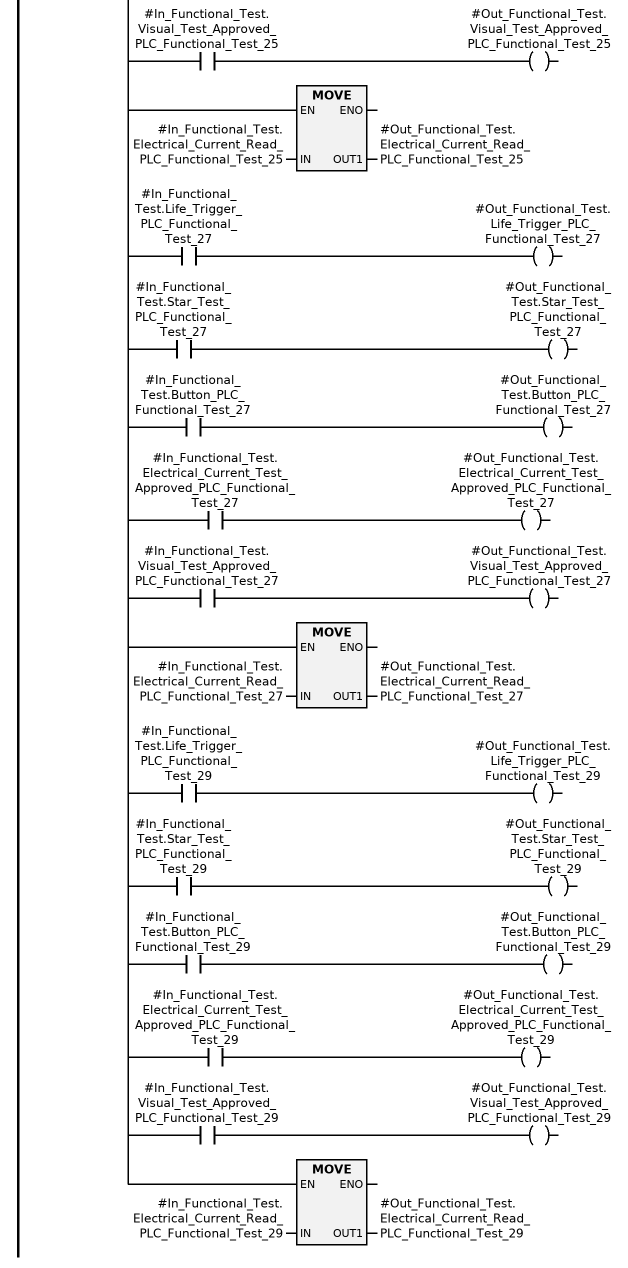
   RUNG wire#powerrail
      { S7_Templates := "SrcType := SInt" } EQ_Contact(in1 := #Test_Station, in2 := 7)
      wire#w1
      Contact( #Life_Trigger )
      Coil( #Out_Functional_Test.Life_Trigger_PLC_Functional_Test_7 )
   END_RUNG
   RUNG wire#w1
      Contact( #Star_Test )
      Coil( #Out_Functional_Test.Star_Test_PLC_Functional_Test_7 )
   END_RUNG
   RUNG wire#w1
      Contact( #Button_Start_Approve )
      Coil( #Out_Functional_Test.Button_PLC_Functional_Test_7 )
   END_RUNG
   RUNG wire#w1
      Contact( #Electrical_Current_Test_Approved )
      Coil( #Out_Functional_Test.Electrical_Current_Test_Approved_PLC_Functional_Test_7 )
   END_RUNG
   RUNG wire#w1
      Contact( #Visual_Test_Approved )
      Coil( #Out_Functional_Test.Visual_Test_Approved_PLC_Functional_Test_7 )
   END_RUNG
   RUNG wire#w1
      Contact( #In_Test_Parameters.Reset_PLC_Functional_Test_7 )
      Coil( #Reset_Functional_Test )
   END_RUNG
   RUNG wire#w1
      Move(in := #Electrical_Current_Read, out1 => #Out_Functional_Test.Electrical_Current_Read_PLC_Functional_Test_7)
   END_RUNG
   RUNG wire#w1
      Contact( #In_Functional_Test.Life_Trigger_PLC_Functional_Test_9 )
      Coil( #Out_Functional_Test.Life_Trigger_PLC_Functional_Test_9 )
   END_RUNG
   RUNG wire#w1
      Contact( #In_Functional_Test.Star_Test_PLC_Functional_Test_9 )
      Coil( #Out_Functional_Test.Star_Test_PLC_Functional_Test_9 )
   END_RUNG
   RUNG wire#w1
      Contact( #In_Functional_Test.Button_PLC_Functional_Test_9 )
      Coil( #Out_Functional_Test.Button_PLC_Functional_Test_9 )
   END_RUNG
   RUNG wire#w1
      Contact( #In_Functional_Test.Electrical_Current_Test_Approved_PLC_Functional_Test_9 )
      Coil( #Out_Functional_Test.Electrical_Current_Test_Approved_PLC_Functional_Test_9 )
   END_RUNG
   RUNG wire#w1
      Contact( #In_Functional_Test.Visual_Test_Approved_PLC_Functional_Test_9 )
      Coil( #Out_Functional_Test.Visual_Test_Approved_PLC_Functional_Test_9 )
   END_RUNG
   RUNG wire#w1
      Move(in := #In_Functional_Test.Electrical_Current_Read_PLC_Functional_Test_9, out1 => #Out_Functional_Test.Electrical_Current_Read_PLC_Functional_Test_9)
   END_RUNG
   RUNG wire#w1
      Contact( #In_Functional_Test.Life_Trigger_PLC_Functional_Test_11 )
      Coil( #Out_Functional_Test.Life_Trigger_PLC_Functional_Test_11 )
   END_RUNG
   RUNG wire#w1
      Contact( #In_Functional_Test.Star_Test_PLC_Functional_Test_11 )
      Coil( #Out_Functional_Test.Star_Test_PLC_Functional_Test_11 )
   END_RUNG
   RUNG wire#w1
      Contact( #In_Functional_Test.Button_PLC_Functional_Test_11 )
      Coil( #Out_Functional_Test.Button_PLC_Functional_Test_11 )
   END_RUNG
   RUNG wire#w1
      Contact( #In_Functional_Test.Electrical_Current_Test_Approved_PLC_Functional_Test_11 )
      Coil( #Out_Functional_Test.Electrical_Current_Test_Approved_PLC_Functional_Test_11 )
   END_RUNG
   RUNG wire#w1
      Contact( #In_Functional_Test.Visual_Test_Approved_PLC_Functional_Test_11 )
      Coil( #Out_Functional_Test.Visual_Test_Approved_PLC_Functional_Test_11 )
   END_RUNG
   RUNG wire#w1
      Move(in := #In_Functional_Test.Electrical_Current_Read_PLC_Functional_Test_11, out1 => #Out_Functional_Test.Electrical_Current_Read_PLC_Functional_Test_11)
   END_RUNG
   RUNG wire#w1
      Contact( #In_Functional_Test.Life_Trigger_PLC_Functional_Test_13 )
      Coil( #Out_Functional_Test.Life_Trigger_PLC_Functional_Test_13 )
   END_RUNG
   RUNG wire#w1
      Contact( #In_Functional_Test.Star_Test_PLC_Functional_Test_13 )
      Coil( #Out_Functional_Test.Star_Test_PLC_Functional_Test_13 )
   END_RUNG
   RUNG wire#w1
      Contact( #In_Functional_Test.Button_PLC_Functional_Test_13 )
      Coil( #Out_Functional_Test.Button_PLC_Functional_Test_13 )
   END_RUNG
   RUNG wire#w1
      Contact( #In_Functional_Test.Electrical_Current_Test_Approved_PLC_Functional_Test_13 )
      Coil( #Out_Functional_Test.Electrical_Current_Test_Approved_PLC_Functional_Test_13 )
   END_RUNG
   RUNG wire#w1
      Contact( #In_Functional_Test.Visual_Test_Approved_PLC_Functional_Test_13 )
      Coil( #Out_Functional_Test.Visual_Test_Approved_PLC_Functional_Test_13 )
   END_RUNG
   RUNG wire#w1
      Move(in := #In_Functional_Test.Electrical_Current_Read_PLC_Functional_Test_13, out1 => #Out_Functional_Test.Electrical_Current_Read_PLC_Functional_Test_13)
   END_RUNG
   RUNG wire#w1
      Contact( #In_Functional_Test.Life_Trigger_PLC_Functional_Test_15 )
      Coil( #Out_Functional_Test.Life_Trigger_PLC_Functional_Test_15 )
   END_RUNG
   RUNG wire#w1
      Contact( #In_Functional_Test.Star_Test_PLC_Functional_Test_15 )
      Coil( #Out_Functional_Test.Star_Test_PLC_Functional_Test_15 )
   END_RUNG
   RUNG wire#w1
      Contact( #In_Functional_Test.Button_PLC_Functional_Test_15 )
      Coil( #Out_Functional_Test.Button_PLC_Functional_Test_15 )
   END_RUNG
   RUNG wire#w1
      Contact( #In_Functional_Test.Electrical_Current_Test_Approved_PLC_Functional_Test_15 )
      Coil( #Out_Functional_Test.Electrical_Current_Test_Approved_PLC_Functional_Test_15 )
   END_RUNG
   RUNG wire#w1
      Contact( #In_Functional_Test.Visual_Test_Approved_PLC_Functional_Test_15 )
      Coil( #Out_Functional_Test.Visual_Test_Approved_PLC_Functional_Test_15 )
   END_RUNG
   RUNG wire#w1
      Move(in := #In_Functional_Test.Electrical_Current_Read_PLC_Functional_Test_15, out1 => #Out_Functional_Test.Electrical_Current_Read_PLC_Functional_Test_15)
   END_RUNG
   RUNG wire#w1
      Contact( #In_Functional_Test.Life_Trigger_PLC_Functional_Test_17 )
      Coil( #Out_Functional_Test.Life_Trigger_PLC_Functional_Test_17 )
   END_RUNG
   RUNG wire#w1
      Contact( #In_Functional_Test.Star_Test_PLC_Functional_Test_17 )
      Coil( #Out_Functional_Test.Star_Test_PLC_Functional_Test_17 )
   END_RUNG
   RUNG wire#w1
      Contact( #In_Functional_Test.Button_PLC_Functional_Test_17 )
      Coil( #Out_Functional_Test.Button_PLC_Functional_Test_17 )
   END_RUNG
   RUNG wire#w1
      Contact( #In_Functional_Test.Electrical_Current_Test_Approved_PLC_Functional_Test_17 )
      Coil( #Out_Functional_Test.Electrical_Current_Test_Approved_PLC_Functional_Test_17 )
   END_RUNG
   RUNG wire#w1
      Contact( #In_Functional_Test.Visual_Test_Approved_PLC_Functional_Test_17 )
      Coil( #Out_Functional_Test.Visual_Test_Approved_PLC_Functional_Test_17 )
   END_RUNG
   RUNG wire#w1
      Move(in := #In_Functional_Test.Electrical_Current_Read_PLC_Functional_Test_17, out1 => #Out_Functional_Test.Electrical_Current_Read_PLC_Functional_Test_17)
   END_RUNG
   RUNG wire#w1
      Contact( #In_Functional_Test.Life_Trigger_PLC_Functional_Test_19 )
      Coil( #Out_Functional_Test.Life_Trigger_PLC_Functional_Test_19 )
   END_RUNG
   RUNG wire#w1
      Contact( #In_Functional_Test.Star_Test_PLC_Functional_Test_19 )
      Coil( #Out_Functional_Test.Star_Test_PLC_Functional_Test_19 )
   END_RUNG
   RUNG wire#w1
      Contact( #In_Functional_Test.Button_PLC_Functional_Test_19 )
      Coil( #Out_Functional_Test.Button_PLC_Functional_Test_19 )
   END_RUNG
   RUNG wire#w1
      Contact( #In_Functional_Test.Electrical_Current_Test_Approved_PLC_Functional_Test_19 )
      Coil( #Out_Functional_Test.Electrical_Current_Test_Approved_PLC_Functional_Test_19 )
   END_RUNG
   RUNG wire#w1
      Contact( #In_Functional_Test.Visual_Test_Approved_PLC_Functional_Test_19 )
      Coil( #Out_Functional_Test.Visual_Test_Approved_PLC_Functional_Test_19 )
   END_RUNG
   RUNG wire#w1
      Move(in := #In_Functional_Test.Electrical_Current_Read_PLC_Functional_Test_19, out1 => #Out_Functional_Test.Electrical_Current_Read_PLC_Functional_Test_19)
   END_RUNG
   RUNG wire#w1
      Contact( #In_Functional_Test.Life_Trigger_PLC_Functional_Test_21 )
      Coil( #Out_Functional_Test.Life_Trigger_PLC_Functional_Test_21 )
   END_RUNG
   RUNG wire#w1
      Contact( #In_Functional_Test.Star_Test_PLC_Functional_Test_21 )
      Coil( #Out_Functional_Test.Star_Test_PLC_Functional_Test_21 )
   END_RUNG
   RUNG wire#w1
      Contact( #In_Functional_Test.Button_PLC_Functional_Test_21 )
      Coil( #Out_Functional_Test.Button_PLC_Functional_Test_21 )
   END_RUNG
   RUNG wire#w1
      Contact( #In_Functional_Test.Electrical_Current_Test_Approved_PLC_Functional_Test_21 )
      Coil( #Out_Functional_Test.Electrical_Current_Test_Approved_PLC_Functional_Test_21 )
   END_RUNG
   RUNG wire#w1
      Contact( #In_Functional_Test.Visual_Test_Approved_PLC_Functional_Test_21 )
      Coil( #Out_Functional_Test.Visual_Test_Approved_PLC_Functional_Test_21 )
   END_RUNG
   RUNG wire#w1
      Move(in := #In_Functional_Test.Electrical_Current_Read_PLC_Functional_Test_21, out1 => #Out_Functional_Test.Electrical_Current_Read_PLC_Functional_Test_21)
   END_RUNG
   RUNG wire#w1
      Contact( #In_Functional_Test.Life_Trigger_PLC_Functional_Test_23 )
      Coil( #Out_Functional_Test.Life_Trigger_PLC_Functional_Test_23 )
   END_RUNG
   RUNG wire#w1
      Contact( #In_Functional_Test.Star_Test_PLC_Functional_Test_23 )
      Coil( #Out_Functional_Test.Star_Test_PLC_Functional_Test_23 )
   END_RUNG
   RUNG wire#w1
      Contact( #In_Functional_Test.Button_PLC_Functional_Test_23 )
      Coil( #Out_Functional_Test.Button_PLC_Functional_Test_23 )
   END_RUNG
   RUNG wire#w1
      Contact( #In_Functional_Test.Electrical_Current_Test_Approved_PLC_Functional_Test_23 )
      Coil( #Out_Functional_Test.Electrical_Current_Test_Approved_PLC_Functional_Test_23 )
   END_RUNG
   RUNG wire#w1
      Contact( #In_Functional_Test.Visual_Test_Approved_PLC_Functional_Test_23 )
      Coil( #Out_Functional_Test.Visual_Test_Approved_PLC_Functional_Test_23 )
   END_RUNG
   RUNG wire#w1
      Move(in := #In_Functional_Test.Electrical_Current_Read_PLC_Functional_Test_23, out1 => #Out_Functional_Test.Electrical_Current_Read_PLC_Functional_Test_23)
   END_RUNG
   RUNG wire#w1
      Contact( #In_Functional_Test.Life_Trigger_PLC_Functional_Test_25 )
      Coil( #Out_Functional_Test.Life_Trigger_PLC_Functional_Test_25 )
   END_RUNG
   RUNG wire#w1
      Contact( #In_Functional_Test.Star_Test_PLC_Functional_Test_25 )
      Coil( #Out_Functional_Test.Star_Test_PLC_Functional_Test_25 )
   END_RUNG
   RUNG wire#w1
      Contact( #In_Functional_Test.Button_PLC_Functional_Test_25 )
      Coil( #Out_Functional_Test.Button_PLC_Functional_Test_25 )
   END_RUNG
   RUNG wire#w1
      Contact( #In_Functional_Test.Electrical_Current_Test_Approved_PLC_Functional_Test_25 )
      Coil( #Out_Functional_Test.Electrical_Current_Test_Approved_PLC_Functional_Test_25 )
   END_RUNG
   RUNG wire#w1
      Contact( #In_Functional_Test.Visual_Test_Approved_PLC_Functional_Test_25 )
      Coil( #Out_Functional_Test.Visual_Test_Approved_PLC_Functional_Test_25 )
   END_RUNG
   RUNG wire#w1
      Move(in := #In_Functional_Test.Electrical_Current_Read_PLC_Functional_Test_25, out1 => #Out_Functional_Test.Electrical_Current_Read_PLC_Functional_Test_25)
   END_RUNG
   RUNG wire#w1
      Contact( #In_Functional_Test.Life_Trigger_PLC_Functional_Test_27 )
      Coil( #Out_Functional_Test.Life_Trigger_PLC_Functional_Test_27 )
   END_RUNG
   RUNG wire#w1
      Contact( #In_Functional_Test.Star_Test_PLC_Functional_Test_27 )
      Coil( #Out_Functional_Test.Star_Test_PLC_Functional_Test_27 )
   END_RUNG
   RUNG wire#w1
      Contact( #In_Functional_Test.Button_PLC_Functional_Test_27 )
      Coil( #Out_Functional_Test.Button_PLC_Functional_Test_27 )
   END_RUNG
   RUNG wire#w1
      Contact( #In_Functional_Test.Electrical_Current_Test_Approved_PLC_Functional_Test_27 )
      Coil( #Out_Functional_Test.Electrical_Current_Test_Approved_PLC_Functional_Test_27 )
   END_RUNG
   RUNG wire#w1
      Contact( #In_Functional_Test.Visual_Test_Approved_PLC_Functional_Test_27 )
      Coil( #Out_Functional_Test.Visual_Test_Approved_PLC_Functional_Test_27 )
   END_RUNG
   RUNG wire#w1
      Move(in := #In_Functional_Test.Electrical_Current_Read_PLC_Functional_Test_27, out1 => #Out_Functional_Test.Electrical_Current_Read_PLC_Functional_Test_27)
   END_RUNG
   RUNG wire#w1
      Contact( #In_Functional_Test.Life_Trigger_PLC_Functional_Test_29 )
      Coil( #Out_Functional_Test.Life_Trigger_PLC_Functional_Test_29 )
   END_RUNG
   RUNG wire#w1
      Contact( #In_Functional_Test.Star_Test_PLC_Functional_Test_29 )
      Coil( #Out_Functional_Test.Star_Test_PLC_Functional_Test_29 )
   END_RUNG
   RUNG wire#w1
      Contact( #In_Functional_Test.Button_PLC_Functional_Test_29 )
      Coil( #Out_Functional_Test.Button_PLC_Functional_Test_29 )
   END_RUNG
   RUNG wire#w1
      Contact( #In_Functional_Test.Electrical_Current_Test_Approved_PLC_Functional_Test_29 )
      Coil( #Out_Functional_Test.Electrical_Current_Test_Approved_PLC_Functional_Test_29 )
   END_RUNG
   RUNG wire#w1
      Contact( #In_Functional_Test.Visual_Test_Approved_PLC_Functional_Test_29 )
      Coil( #Out_Functional_Test.Visual_Test_Approved_PLC_Functional_Test_29 )
   END_RUNG
   RUNG wire#w1
      Move(in := #In_Functional_Test.Electrical_Current_Read_PLC_Functional_Test_29, out1 => #Out_Functional_Test.Electrical_Current_Read_PLC_Functional_Test_29)
   END_RUNG
   // the same network as SCL:
   #_w1 := #Test_Station = 7;
   #Out_Functional_Test.Life_Trigger_PLC_Functional_Test_7 := #_w1 AND #Life_Trigger;
   #Out_Functional_Test.Star_Test_PLC_Functional_Test_7 := #_w1 AND #Star_Test;
   #Out_Functional_Test.Button_PLC_Functional_Test_7 := #_w1 AND #Button_Start_Approve;
   #Out_Functional_Test.Electrical_Current_Test_Approved_PLC_Functional_Test_7 := #_w1 AND #Electrical_Current_Test_Approved;
   #Out_Functional_Test.Visual_Test_Approved_PLC_Functional_Test_7 := #_w1 AND #Visual_Test_Approved;
   #Reset_Functional_Test := #_w1 AND #In_Test_Parameters.Reset_PLC_Functional_Test_7;
   IF #_w1 THEN
       #Out_Functional_Test.Electrical_Current_Read_PLC_Functional_Test_7 := #Electrical_Current_Read;
   END_IF;
   #Out_Functional_Test.Life_Trigger_PLC_Functional_Test_9 := #_w1 AND #In_Functional_Test.Life_Trigger_PLC_Functional_Test_9;
   #Out_Functional_Test.Star_Test_PLC_Functional_Test_9 := #_w1 AND #In_Functional_Test.Star_Test_PLC_Functional_Test_9;
   #Out_Functional_Test.Button_PLC_Functional_Test_9 := #_w1 AND #In_Functional_Test.Button_PLC_Functional_Test_9;
   #Out_Functional_Test.Electrical_Current_Test_Approved_PLC_Functional_Test_9 := #_w1 AND #In_Functional_Test.Electrical_Current_Test_Approved_PLC_Functional_Test_9;
   #Out_Functional_Test.Visual_Test_Approved_PLC_Functional_Test_9 := #_w1 AND #In_Functional_Test.Visual_Test_Approved_PLC_Functional_Test_9;
   IF #_w1 THEN
       #Out_Functional_Test.Electrical_Current_Read_PLC_Functional_Test_9 := #In_Functional_Test.Electrical_Current_Read_PLC_Functional_Test_9;
   END_IF;
   #Out_Functional_Test.Life_Trigger_PLC_Functional_Test_11 := #_w1 AND #In_Functional_Test.Life_Trigger_PLC_Functional_Test_11;
   #Out_Functional_Test.Star_Test_PLC_Functional_Test_11 := #_w1 AND #In_Functional_Test.Star_Test_PLC_Functional_Test_11;
   #Out_Functional_Test.Button_PLC_Functional_Test_11 := #_w1 AND #In_Functional_Test.Button_PLC_Functional_Test_11;
   #Out_Functional_Test.Electrical_Current_Test_Approved_PLC_Functional_Test_11 := #_w1 AND #In_Functional_Test.Electrical_Current_Test_Approved_PLC_Functional_Test_11;
   #Out_Functional_Test.Visual_Test_Approved_PLC_Functional_Test_11 := #_w1 AND #In_Functional_Test.Visual_Test_Approved_PLC_Functional_Test_11;
   IF #_w1 THEN
       #Out_Functional_Test.Electrical_Current_Read_PLC_Functional_Test_11 := #In_Functional_Test.Electrical_Current_Read_PLC_Functional_Test_11;
   END_IF;
   #Out_Functional_Test.Life_Trigger_PLC_Functional_Test_13 := #_w1 AND #In_Functional_Test.Life_Trigger_PLC_Functional_Test_13;
   #Out_Functional_Test.Star_Test_PLC_Functional_Test_13 := #_w1 AND #In_Functional_Test.Star_Test_PLC_Functional_Test_13;
   #Out_Functional_Test.Button_PLC_Functional_Test_13 := #_w1 AND #In_Functional_Test.Button_PLC_Functional_Test_13;
   #Out_Functional_Test.Electrical_Current_Test_Approved_PLC_Functional_Test_13 := #_w1 AND #In_Functional_Test.Electrical_Current_Test_Approved_PLC_Functional_Test_13;
   #Out_Functional_Test.Visual_Test_Approved_PLC_Functional_Test_13 := #_w1 AND #In_Functional_Test.Visual_Test_Approved_PLC_Functional_Test_13;
   IF #_w1 THEN
       #Out_Functional_Test.Electrical_Current_Read_PLC_Functional_Test_13 := #In_Functional_Test.Electrical_Current_Read_PLC_Functional_Test_13;
   END_IF;
   #Out_Functional_Test.Life_Trigger_PLC_Functional_Test_15 := #_w1 AND #In_Functional_Test.Life_Trigger_PLC_Functional_Test_15;
   #Out_Functional_Test.Star_Test_PLC_Functional_Test_15 := #_w1 AND #In_Functional_Test.Star_Test_PLC_Functional_Test_15;
   #Out_Functional_Test.Button_PLC_Functional_Test_15 := #_w1 AND #In_Functional_Test.Button_PLC_Functional_Test_15;
   #Out_Functional_Test.Electrical_Current_Test_Approved_PLC_Functional_Test_15 := #_w1 AND #In_Functional_Test.Electrical_Current_Test_Approved_PLC_Functional_Test_15;
   #Out_Functional_Test.Visual_Test_Approved_PLC_Functional_Test_15 := #_w1 AND #In_Functional_Test.Visual_Test_Approved_PLC_Functional_Test_15;
   IF #_w1 THEN
       #Out_Functional_Test.Electrical_Current_Read_PLC_Functional_Test_15 := #In_Functional_Test.Electrical_Current_Read_PLC_Functional_Test_15;
   END_IF;
   #Out_Functional_Test.Life_Trigger_PLC_Functional_Test_17 := #_w1 AND #In_Functional_Test.Life_Trigger_PLC_Functional_Test_17;
   #Out_Functional_Test.Star_Test_PLC_Functional_Test_17 := #_w1 AND #In_Functional_Test.Star_Test_PLC_Functional_Test_17;
   #Out_Functional_Test.Button_PLC_Functional_Test_17 := #_w1 AND #In_Functional_Test.Button_PLC_Functional_Test_17;
   #Out_Functional_Test.Electrical_Current_Test_Approved_PLC_Functional_Test_17 := #_w1 AND #In_Functional_Test.Electrical_Current_Test_Approved_PLC_Functional_Test_17;
   #Out_Functional_Test.Visual_Test_Approved_PLC_Functional_Test_17 := #_w1 AND #In_Functional_Test.Visual_Test_Approved_PLC_Functional_Test_17;
   IF #_w1 THEN
       #Out_Functional_Test.Electrical_Current_Read_PLC_Functional_Test_17 := #In_Functional_Test.Electrical_Current_Read_PLC_Functional_Test_17;
   END_IF;
   #Out_Functional_Test.Life_Trigger_PLC_Functional_Test_19 := #_w1 AND #In_Functional_Test.Life_Trigger_PLC_Functional_Test_19;
   #Out_Functional_Test.Star_Test_PLC_Functional_Test_19 := #_w1 AND #In_Functional_Test.Star_Test_PLC_Functional_Test_19;
   #Out_Functional_Test.Button_PLC_Functional_Test_19 := #_w1 AND #In_Functional_Test.Button_PLC_Functional_Test_19;
   #Out_Functional_Test.Electrical_Current_Test_Approved_PLC_Functional_Test_19 := #_w1 AND #In_Functional_Test.Electrical_Current_Test_Approved_PLC_Functional_Test_19;
   #Out_Functional_Test.Visual_Test_Approved_PLC_Functional_Test_19 := #_w1 AND #In_Functional_Test.Visual_Test_Approved_PLC_Functional_Test_19;
   IF #_w1 THEN
       #Out_Functional_Test.Electrical_Current_Read_PLC_Functional_Test_19 := #In_Functional_Test.Electrical_Current_Read_PLC_Functional_Test_19;
   END_IF;
   #Out_Functional_Test.Life_Trigger_PLC_Functional_Test_21 := #_w1 AND #In_Functional_Test.Life_Trigger_PLC_Functional_Test_21;
   #Out_Functional_Test.Star_Test_PLC_Functional_Test_21 := #_w1 AND #In_Functional_Test.Star_Test_PLC_Functional_Test_21;
   #Out_Functional_Test.Button_PLC_Functional_Test_21 := #_w1 AND #In_Functional_Test.Button_PLC_Functional_Test_21;
   #Out_Functional_Test.Electrical_Current_Test_Approved_PLC_Functional_Test_21 := #_w1 AND #In_Functional_Test.Electrical_Current_Test_Approved_PLC_Functional_Test_21;
   #Out_Functional_Test.Visual_Test_Approved_PLC_Functional_Test_21 := #_w1 AND #In_Functional_Test.Visual_Test_Approved_PLC_Functional_Test_21;
   IF #_w1 THEN
       #Out_Functional_Test.Electrical_Current_Read_PLC_Functional_Test_21 := #In_Functional_Test.Electrical_Current_Read_PLC_Functional_Test_21;
   END_IF;
   #Out_Functional_Test.Life_Trigger_PLC_Functional_Test_23 := #_w1 AND #In_Functional_Test.Life_Trigger_PLC_Functional_Test_23;
   #Out_Functional_Test.Star_Test_PLC_Functional_Test_23 := #_w1 AND #In_Functional_Test.Star_Test_PLC_Functional_Test_23;
   #Out_Functional_Test.Button_PLC_Functional_Test_23 := #_w1 AND #In_Functional_Test.Button_PLC_Functional_Test_23;
   #Out_Functional_Test.Electrical_Current_Test_Approved_PLC_Functional_Test_23 := #_w1 AND #In_Functional_Test.Electrical_Current_Test_Approved_PLC_Functional_Test_23;
   #Out_Functional_Test.Visual_Test_Approved_PLC_Functional_Test_23 := #_w1 AND #In_Functional_Test.Visual_Test_Approved_PLC_Functional_Test_23;
   IF #_w1 THEN
       #Out_Functional_Test.Electrical_Current_Read_PLC_Functional_Test_23 := #In_Functional_Test.Electrical_Current_Read_PLC_Functional_Test_23;
   END_IF;
   #Out_Functional_Test.Life_Trigger_PLC_Functional_Test_25 := #_w1 AND #In_Functional_Test.Life_Trigger_PLC_Functional_Test_25;
   #Out_Functional_Test.Star_Test_PLC_Functional_Test_25 := #_w1 AND #In_Functional_Test.Star_Test_PLC_Functional_Test_25;
   #Out_Functional_Test.Button_PLC_Functional_Test_25 := #_w1 AND #In_Functional_Test.Button_PLC_Functional_Test_25;
   #Out_Functional_Test.Electrical_Current_Test_Approved_PLC_Functional_Test_25 := #_w1 AND #In_Functional_Test.Electrical_Current_Test_Approved_PLC_Functional_Test_25;
   #Out_Functional_Test.Visual_Test_Approved_PLC_Functional_Test_25 := #_w1 AND #In_Functional_Test.Visual_Test_Approved_PLC_Functional_Test_25;
   IF #_w1 THEN
       #Out_Functional_Test.Electrical_Current_Read_PLC_Functional_Test_25 := #In_Functional_Test.Electrical_Current_Read_PLC_Functional_Test_25;
   END_IF;
   #Out_Functional_Test.Life_Trigger_PLC_Functional_Test_27 := #_w1 AND #In_Functional_Test.Life_Trigger_PLC_Functional_Test_27;
   #Out_Functional_Test.Star_Test_PLC_Functional_Test_27 := #_w1 AND #In_Functional_Test.Star_Test_PLC_Functional_Test_27;
   #Out_Functional_Test.Button_PLC_Functional_Test_27 := #_w1 AND #In_Functional_Test.Button_PLC_Functional_Test_27;
   #Out_Functional_Test.Electrical_Current_Test_Approved_PLC_Functional_Test_27 := #_w1 AND #In_Functional_Test.Electrical_Current_Test_Approved_PLC_Functional_Test_27;
   #Out_Functional_Test.Visual_Test_Approved_PLC_Functional_Test_27 := #_w1 AND #In_Functional_Test.Visual_Test_Approved_PLC_Functional_Test_27;
   IF #_w1 THEN
       #Out_Functional_Test.Electrical_Current_Read_PLC_Functional_Test_27 := #In_Functional_Test.Electrical_Current_Read_PLC_Functional_Test_27;
   END_IF;
   #Out_Functional_Test.Life_Trigger_PLC_Functional_Test_29 := #_w1 AND #In_Functional_Test.Life_Trigger_PLC_Functional_Test_29;
   #Out_Functional_Test.Star_Test_PLC_Functional_Test_29 := #_w1 AND #In_Functional_Test.Star_Test_PLC_Functional_Test_29;
   #Out_Functional_Test.Button_PLC_Functional_Test_29 := #_w1 AND #In_Functional_Test.Button_PLC_Functional_Test_29;
   #Out_Functional_Test.Electrical_Current_Test_Approved_PLC_Functional_Test_29 := #_w1 AND #In_Functional_Test.Electrical_Current_Test_Approved_PLC_Functional_Test_29;
   #Out_Functional_Test.Visual_Test_Approved_PLC_Functional_Test_29 := #_w1 AND #In_Functional_Test.Visual_Test_Approved_PLC_Functional_Test_29;
   IF #_w1 THEN
       #Out_Functional_Test.Electrical_Current_Read_PLC_Functional_Test_29 := #In_Functional_Test.Electrical_Current_Read_PLC_Functional_Test_29;
   END_IF;
END_REGION

REGION Network 6: Functional Test Station 9
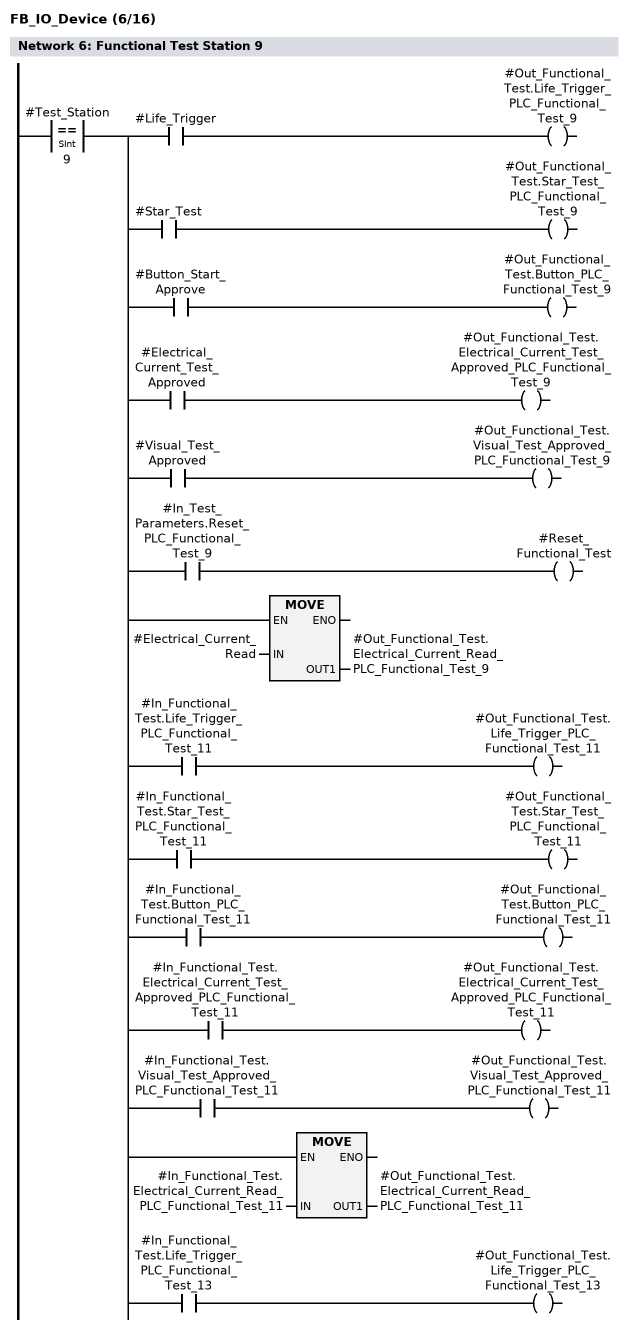
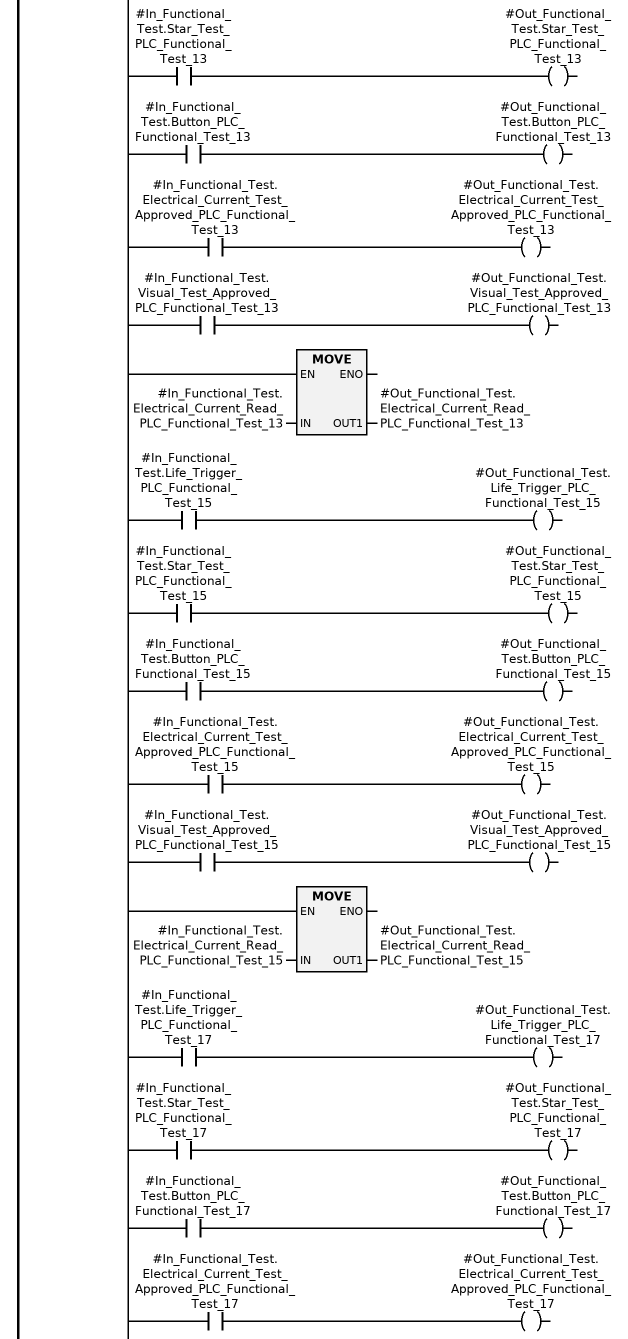
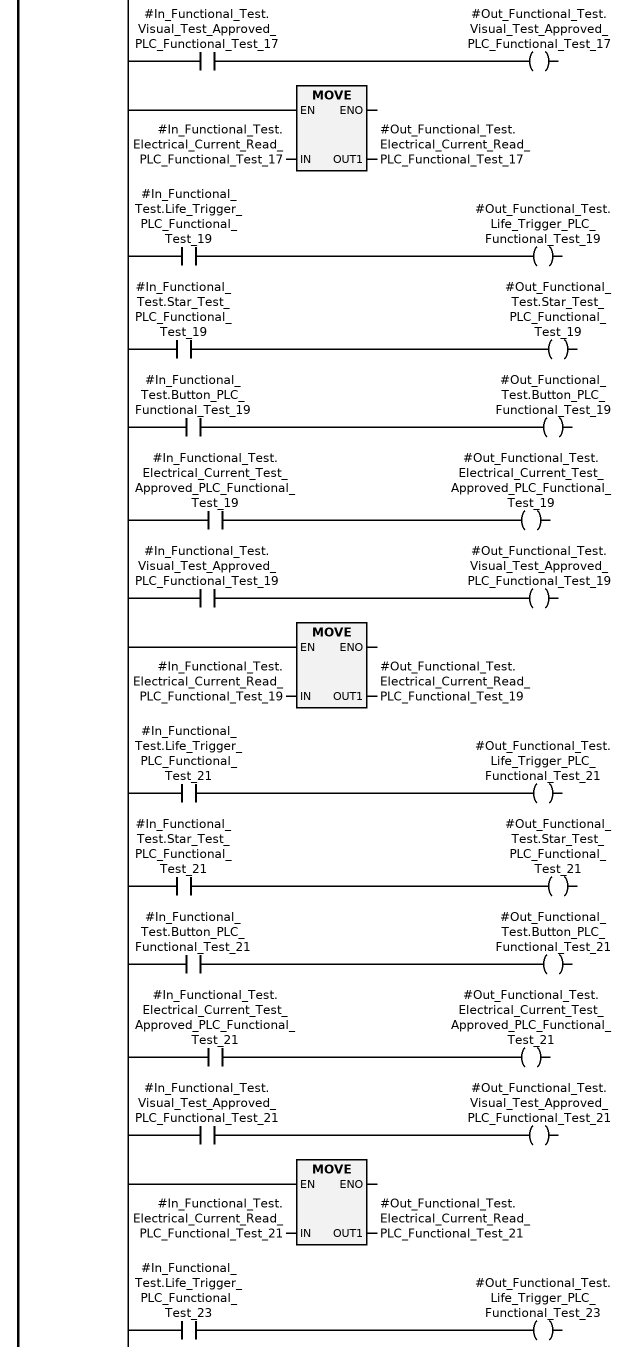
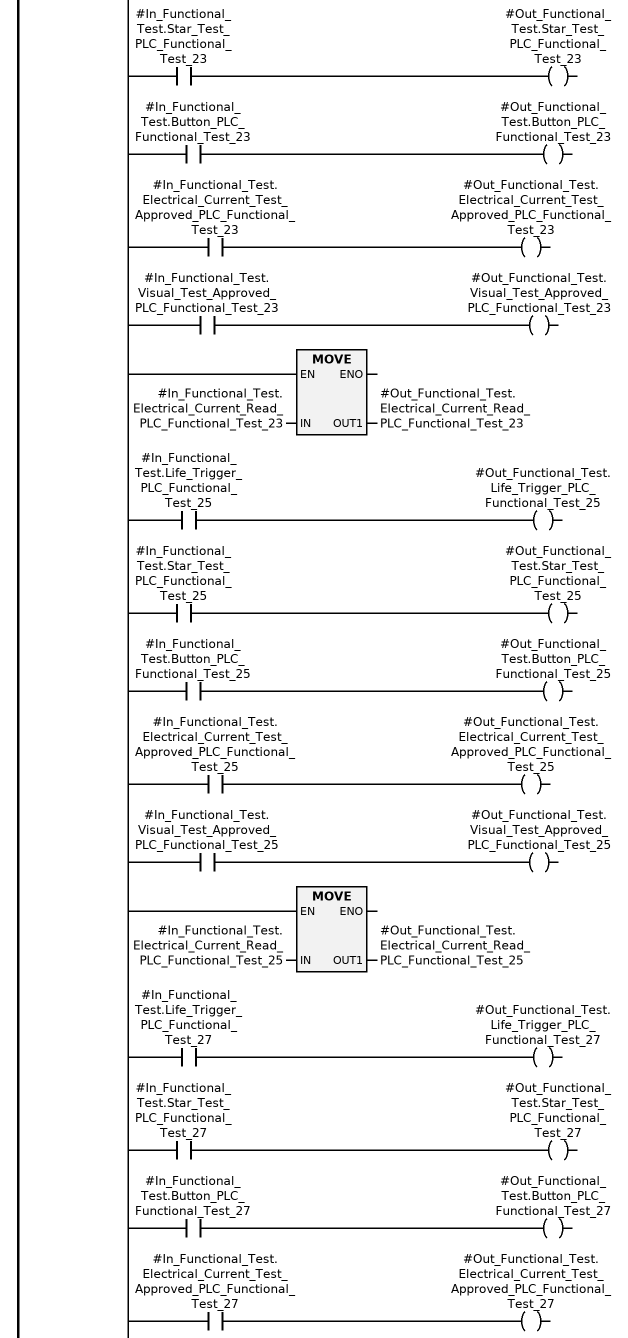
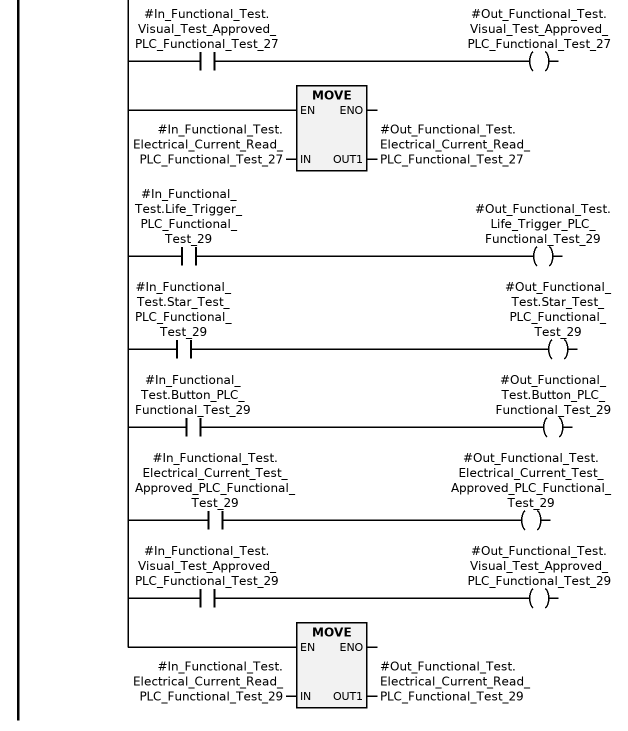
   RUNG wire#powerrail
      { S7_Templates := "SrcType := SInt" } EQ_Contact(in1 := #Test_Station, in2 := 9)
      wire#w1
      Contact( #Life_Trigger )
      Coil( #Out_Functional_Test.Life_Trigger_PLC_Functional_Test_9 )
   END_RUNG
   RUNG wire#w1
      Contact( #Star_Test )
      Coil( #Out_Functional_Test.Star_Test_PLC_Functional_Test_9 )
   END_RUNG
   RUNG wire#w1
      Contact( #Button_Start_Approve )
      Coil( #Out_Functional_Test.Button_PLC_Functional_Test_9 )
   END_RUNG
   RUNG wire#w1
      Contact( #Electrical_Current_Test_Approved )
      Coil( #Out_Functional_Test.Electrical_Current_Test_Approved_PLC_Functional_Test_9 )
   END_RUNG
   RUNG wire#w1
      Contact( #Visual_Test_Approved )
      Coil( #Out_Functional_Test.Visual_Test_Approved_PLC_Functional_Test_9 )
   END_RUNG
   RUNG wire#w1
      Contact( #In_Test_Parameters.Reset_PLC_Functional_Test_9 )
      Coil( #Reset_Functional_Test )
   END_RUNG
   RUNG wire#w1
      Move(in := #Electrical_Current_Read, out1 => #Out_Functional_Test.Electrical_Current_Read_PLC_Functional_Test_9)
   END_RUNG
   RUNG wire#w1
      Contact( #In_Functional_Test.Life_Trigger_PLC_Functional_Test_11 )
      Coil( #Out_Functional_Test.Life_Trigger_PLC_Functional_Test_11 )
   END_RUNG
   RUNG wire#w1
      Contact( #In_Functional_Test.Star_Test_PLC_Functional_Test_11 )
      Coil( #Out_Functional_Test.Star_Test_PLC_Functional_Test_11 )
   END_RUNG
   RUNG wire#w1
      Contact( #In_Functional_Test.Button_PLC_Functional_Test_11 )
      Coil( #Out_Functional_Test.Button_PLC_Functional_Test_11 )
   END_RUNG
   RUNG wire#w1
      Contact( #In_Functional_Test.Electrical_Current_Test_Approved_PLC_Functional_Test_11 )
      Coil( #Out_Functional_Test.Electrical_Current_Test_Approved_PLC_Functional_Test_11 )
   END_RUNG
   RUNG wire#w1
      Contact( #In_Functional_Test.Visual_Test_Approved_PLC_Functional_Test_11 )
      Coil( #Out_Functional_Test.Visual_Test_Approved_PLC_Functional_Test_11 )
   END_RUNG
   RUNG wire#w1
      Move(in := #In_Functional_Test.Electrical_Current_Read_PLC_Functional_Test_11, out1 => #Out_Functional_Test.Electrical_Current_Read_PLC_Functional_Test_11)
   END_RUNG
   RUNG wire#w1
      Contact( #In_Functional_Test.Life_Trigger_PLC_Functional_Test_13 )
      Coil( #Out_Functional_Test.Life_Trigger_PLC_Functional_Test_13 )
   END_RUNG
   RUNG wire#w1
      Contact( #In_Functional_Test.Star_Test_PLC_Functional_Test_13 )
      Coil( #Out_Functional_Test.Star_Test_PLC_Functional_Test_13 )
   END_RUNG
   RUNG wire#w1
      Contact( #In_Functional_Test.Button_PLC_Functional_Test_13 )
      Coil( #Out_Functional_Test.Button_PLC_Functional_Test_13 )
   END_RUNG
   RUNG wire#w1
      Contact( #In_Functional_Test.Electrical_Current_Test_Approved_PLC_Functional_Test_13 )
      Coil( #Out_Functional_Test.Electrical_Current_Test_Approved_PLC_Functional_Test_13 )
   END_RUNG
   RUNG wire#w1
      Contact( #In_Functional_Test.Visual_Test_Approved_PLC_Functional_Test_13 )
      Coil( #Out_Functional_Test.Visual_Test_Approved_PLC_Functional_Test_13 )
   END_RUNG
   RUNG wire#w1
      Move(in := #In_Functional_Test.Electrical_Current_Read_PLC_Functional_Test_13, out1 => #Out_Functional_Test.Electrical_Current_Read_PLC_Functional_Test_13)
   END_RUNG
   RUNG wire#w1
      Contact( #In_Functional_Test.Life_Trigger_PLC_Functional_Test_15 )
      Coil( #Out_Functional_Test.Life_Trigger_PLC_Functional_Test_15 )
   END_RUNG
   RUNG wire#w1
      Contact( #In_Functional_Test.Star_Test_PLC_Functional_Test_15 )
      Coil( #Out_Functional_Test.Star_Test_PLC_Functional_Test_15 )
   END_RUNG
   RUNG wire#w1
      Contact( #In_Functional_Test.Button_PLC_Functional_Test_15 )
      Coil( #Out_Functional_Test.Button_PLC_Functional_Test_15 )
   END_RUNG
   RUNG wire#w1
      Contact( #In_Functional_Test.Electrical_Current_Test_Approved_PLC_Functional_Test_15 )
      Coil( #Out_Functional_Test.Electrical_Current_Test_Approved_PLC_Functional_Test_15 )
   END_RUNG
   RUNG wire#w1
      Contact( #In_Functional_Test.Visual_Test_Approved_PLC_Functional_Test_15 )
      Coil( #Out_Functional_Test.Visual_Test_Approved_PLC_Functional_Test_15 )
   END_RUNG
   RUNG wire#w1
      Move(in := #In_Functional_Test.Electrical_Current_Read_PLC_Functional_Test_15, out1 => #Out_Functional_Test.Electrical_Current_Read_PLC_Functional_Test_15)
   END_RUNG
   RUNG wire#w1
      Contact( #In_Functional_Test.Life_Trigger_PLC_Functional_Test_17 )
      Coil( #Out_Functional_Test.Life_Trigger_PLC_Functional_Test_17 )
   END_RUNG
   RUNG wire#w1
      Contact( #In_Functional_Test.Star_Test_PLC_Functional_Test_17 )
      Coil( #Out_Functional_Test.Star_Test_PLC_Functional_Test_17 )
   END_RUNG
   RUNG wire#w1
      Contact( #In_Functional_Test.Button_PLC_Functional_Test_17 )
      Coil( #Out_Functional_Test.Button_PLC_Functional_Test_17 )
   END_RUNG
   RUNG wire#w1
      Contact( #In_Functional_Test.Electrical_Current_Test_Approved_PLC_Functional_Test_17 )
      Coil( #Out_Functional_Test.Electrical_Current_Test_Approved_PLC_Functional_Test_17 )
   END_RUNG
   RUNG wire#w1
      Contact( #In_Functional_Test.Visual_Test_Approved_PLC_Functional_Test_17 )
      Coil( #Out_Functional_Test.Visual_Test_Approved_PLC_Functional_Test_17 )
   END_RUNG
   RUNG wire#w1
      Move(in := #In_Functional_Test.Electrical_Current_Read_PLC_Functional_Test_17, out1 => #Out_Functional_Test.Electrical_Current_Read_PLC_Functional_Test_17)
   END_RUNG
   RUNG wire#w1
      Contact( #In_Functional_Test.Life_Trigger_PLC_Functional_Test_19 )
      Coil( #Out_Functional_Test.Life_Trigger_PLC_Functional_Test_19 )
   END_RUNG
   RUNG wire#w1
      Contact( #In_Functional_Test.Star_Test_PLC_Functional_Test_19 )
      Coil( #Out_Functional_Test.Star_Test_PLC_Functional_Test_19 )
   END_RUNG
   RUNG wire#w1
      Contact( #In_Functional_Test.Button_PLC_Functional_Test_19 )
      Coil( #Out_Functional_Test.Button_PLC_Functional_Test_19 )
   END_RUNG
   RUNG wire#w1
      Contact( #In_Functional_Test.Electrical_Current_Test_Approved_PLC_Functional_Test_19 )
      Coil( #Out_Functional_Test.Electrical_Current_Test_Approved_PLC_Functional_Test_19 )
   END_RUNG
   RUNG wire#w1
      Contact( #In_Functional_Test.Visual_Test_Approved_PLC_Functional_Test_19 )
      Coil( #Out_Functional_Test.Visual_Test_Approved_PLC_Functional_Test_19 )
   END_RUNG
   RUNG wire#w1
      Move(in := #In_Functional_Test.Electrical_Current_Read_PLC_Functional_Test_19, out1 => #Out_Functional_Test.Electrical_Current_Read_PLC_Functional_Test_19)
   END_RUNG
   RUNG wire#w1
      Contact( #In_Functional_Test.Life_Trigger_PLC_Functional_Test_21 )
      Coil( #Out_Functional_Test.Life_Trigger_PLC_Functional_Test_21 )
   END_RUNG
   RUNG wire#w1
      Contact( #In_Functional_Test.Star_Test_PLC_Functional_Test_21 )
      Coil( #Out_Functional_Test.Star_Test_PLC_Functional_Test_21 )
   END_RUNG
   RUNG wire#w1
      Contact( #In_Functional_Test.Button_PLC_Functional_Test_21 )
      Coil( #Out_Functional_Test.Button_PLC_Functional_Test_21 )
   END_RUNG
   RUNG wire#w1
      Contact( #In_Functional_Test.Electrical_Current_Test_Approved_PLC_Functional_Test_21 )
      Coil( #Out_Functional_Test.Electrical_Current_Test_Approved_PLC_Functional_Test_21 )
   END_RUNG
   RUNG wire#w1
      Contact( #In_Functional_Test.Visual_Test_Approved_PLC_Functional_Test_21 )
      Coil( #Out_Functional_Test.Visual_Test_Approved_PLC_Functional_Test_21 )
   END_RUNG
   RUNG wire#w1
      Move(in := #In_Functional_Test.Electrical_Current_Read_PLC_Functional_Test_21, out1 => #Out_Functional_Test.Electrical_Current_Read_PLC_Functional_Test_21)
   END_RUNG
   RUNG wire#w1
      Contact( #In_Functional_Test.Life_Trigger_PLC_Functional_Test_23 )
      Coil( #Out_Functional_Test.Life_Trigger_PLC_Functional_Test_23 )
   END_RUNG
   RUNG wire#w1
      Contact( #In_Functional_Test.Star_Test_PLC_Functional_Test_23 )
      Coil( #Out_Functional_Test.Star_Test_PLC_Functional_Test_23 )
   END_RUNG
   RUNG wire#w1
      Contact( #In_Functional_Test.Button_PLC_Functional_Test_23 )
      Coil( #Out_Functional_Test.Button_PLC_Functional_Test_23 )
   END_RUNG
   RUNG wire#w1
      Contact( #In_Functional_Test.Electrical_Current_Test_Approved_PLC_Functional_Test_23 )
      Coil( #Out_Functional_Test.Electrical_Current_Test_Approved_PLC_Functional_Test_23 )
   END_RUNG
   RUNG wire#w1
      Contact( #In_Functional_Test.Visual_Test_Approved_PLC_Functional_Test_23 )
      Coil( #Out_Functional_Test.Visual_Test_Approved_PLC_Functional_Test_23 )
   END_RUNG
   RUNG wire#w1
      Move(in := #In_Functional_Test.Electrical_Current_Read_PLC_Functional_Test_23, out1 => #Out_Functional_Test.Electrical_Current_Read_PLC_Functional_Test_23)
   END_RUNG
   RUNG wire#w1
      Contact( #In_Functional_Test.Life_Trigger_PLC_Functional_Test_25 )
      Coil( #Out_Functional_Test.Life_Trigger_PLC_Functional_Test_25 )
   END_RUNG
   RUNG wire#w1
      Contact( #In_Functional_Test.Star_Test_PLC_Functional_Test_25 )
      Coil( #Out_Functional_Test.Star_Test_PLC_Functional_Test_25 )
   END_RUNG
   RUNG wire#w1
      Contact( #In_Functional_Test.Button_PLC_Functional_Test_25 )
      Coil( #Out_Functional_Test.Button_PLC_Functional_Test_25 )
   END_RUNG
   RUNG wire#w1
      Contact( #In_Functional_Test.Electrical_Current_Test_Approved_PLC_Functional_Test_25 )
      Coil( #Out_Functional_Test.Electrical_Current_Test_Approved_PLC_Functional_Test_25 )
   END_RUNG
   RUNG wire#w1
      Contact( #In_Functional_Test.Visual_Test_Approved_PLC_Functional_Test_25 )
      Coil( #Out_Functional_Test.Visual_Test_Approved_PLC_Functional_Test_25 )
   END_RUNG
   RUNG wire#w1
      Move(in := #In_Functional_Test.Electrical_Current_Read_PLC_Functional_Test_25, out1 => #Out_Functional_Test.Electrical_Current_Read_PLC_Functional_Test_25)
   END_RUNG
   RUNG wire#w1
      Contact( #In_Functional_Test.Life_Trigger_PLC_Functional_Test_27 )
      Coil( #Out_Functional_Test.Life_Trigger_PLC_Functional_Test_27 )
   END_RUNG
   RUNG wire#w1
      Contact( #In_Functional_Test.Star_Test_PLC_Functional_Test_27 )
      Coil( #Out_Functional_Test.Star_Test_PLC_Functional_Test_27 )
   END_RUNG
   RUNG wire#w1
      Contact( #In_Functional_Test.Button_PLC_Functional_Test_27 )
      Coil( #Out_Functional_Test.Button_PLC_Functional_Test_27 )
   END_RUNG
   RUNG wire#w1
      Contact( #In_Functional_Test.Electrical_Current_Test_Approved_PLC_Functional_Test_27 )
      Coil( #Out_Functional_Test.Electrical_Current_Test_Approved_PLC_Functional_Test_27 )
   END_RUNG
   RUNG wire#w1
      Contact( #In_Functional_Test.Visual_Test_Approved_PLC_Functional_Test_27 )
      Coil( #Out_Functional_Test.Visual_Test_Approved_PLC_Functional_Test_27 )
   END_RUNG
   RUNG wire#w1
      Move(in := #In_Functional_Test.Electrical_Current_Read_PLC_Functional_Test_27, out1 => #Out_Functional_Test.Electrical_Current_Read_PLC_Functional_Test_27)
   END_RUNG
   RUNG wire#w1
      Contact( #In_Functional_Test.Life_Trigger_PLC_Functional_Test_29 )
      Coil( #Out_Functional_Test.Life_Trigger_PLC_Functional_Test_29 )
   END_RUNG
   RUNG wire#w1
      Contact( #In_Functional_Test.Star_Test_PLC_Functional_Test_29 )
      Coil( #Out_Functional_Test.Star_Test_PLC_Functional_Test_29 )
   END_RUNG
   RUNG wire#w1
      Contact( #In_Functional_Test.Button_PLC_Functional_Test_29 )
      Coil( #Out_Functional_Test.Button_PLC_Functional_Test_29 )
   END_RUNG
   RUNG wire#w1
      Contact( #In_Functional_Test.Electrical_Current_Test_Approved_PLC_Functional_Test_29 )
      Coil( #Out_Functional_Test.Electrical_Current_Test_Approved_PLC_Functional_Test_29 )
   END_RUNG
   RUNG wire#w1
      Contact( #In_Functional_Test.Visual_Test_Approved_PLC_Functional_Test_29 )
      Coil( #Out_Functional_Test.Visual_Test_Approved_PLC_Functional_Test_29 )
   END_RUNG
   RUNG wire#w1
      Move(in := #In_Functional_Test.Electrical_Current_Read_PLC_Functional_Test_29, out1 => #Out_Functional_Test.Electrical_Current_Read_PLC_Functional_Test_29)
   END_RUNG
   // the same network as SCL:
   #_w1 := #Test_Station = 9;
   #Out_Functional_Test.Life_Trigger_PLC_Functional_Test_9 := #_w1 AND #Life_Trigger;
   #Out_Functional_Test.Star_Test_PLC_Functional_Test_9 := #_w1 AND #Star_Test;
   #Out_Functional_Test.Button_PLC_Functional_Test_9 := #_w1 AND #Button_Start_Approve;
   #Out_Functional_Test.Electrical_Current_Test_Approved_PLC_Functional_Test_9 := #_w1 AND #Electrical_Current_Test_Approved;
   #Out_Functional_Test.Visual_Test_Approved_PLC_Functional_Test_9 := #_w1 AND #Visual_Test_Approved;
   #Reset_Functional_Test := #_w1 AND #In_Test_Parameters.Reset_PLC_Functional_Test_9;
   IF #_w1 THEN
       #Out_Functional_Test.Electrical_Current_Read_PLC_Functional_Test_9 := #Electrical_Current_Read;
   END_IF;
   #Out_Functional_Test.Life_Trigger_PLC_Functional_Test_11 := #_w1 AND #In_Functional_Test.Life_Trigger_PLC_Functional_Test_11;
   #Out_Functional_Test.Star_Test_PLC_Functional_Test_11 := #_w1 AND #In_Functional_Test.Star_Test_PLC_Functional_Test_11;
   #Out_Functional_Test.Button_PLC_Functional_Test_11 := #_w1 AND #In_Functional_Test.Button_PLC_Functional_Test_11;
   #Out_Functional_Test.Electrical_Current_Test_Approved_PLC_Functional_Test_11 := #_w1 AND #In_Functional_Test.Electrical_Current_Test_Approved_PLC_Functional_Test_11;
   #Out_Functional_Test.Visual_Test_Approved_PLC_Functional_Test_11 := #_w1 AND #In_Functional_Test.Visual_Test_Approved_PLC_Functional_Test_11;
   IF #_w1 THEN
       #Out_Functional_Test.Electrical_Current_Read_PLC_Functional_Test_11 := #In_Functional_Test.Electrical_Current_Read_PLC_Functional_Test_11;
   END_IF;
   #Out_Functional_Test.Life_Trigger_PLC_Functional_Test_13 := #_w1 AND #In_Functional_Test.Life_Trigger_PLC_Functional_Test_13;
   #Out_Functional_Test.Star_Test_PLC_Functional_Test_13 := #_w1 AND #In_Functional_Test.Star_Test_PLC_Functional_Test_13;
   #Out_Functional_Test.Button_PLC_Functional_Test_13 := #_w1 AND #In_Functional_Test.Button_PLC_Functional_Test_13;
   #Out_Functional_Test.Electrical_Current_Test_Approved_PLC_Functional_Test_13 := #_w1 AND #In_Functional_Test.Electrical_Current_Test_Approved_PLC_Functional_Test_13;
   #Out_Functional_Test.Visual_Test_Approved_PLC_Functional_Test_13 := #_w1 AND #In_Functional_Test.Visual_Test_Approved_PLC_Functional_Test_13;
   IF #_w1 THEN
       #Out_Functional_Test.Electrical_Current_Read_PLC_Functional_Test_13 := #In_Functional_Test.Electrical_Current_Read_PLC_Functional_Test_13;
   END_IF;
   #Out_Functional_Test.Life_Trigger_PLC_Functional_Test_15 := #_w1 AND #In_Functional_Test.Life_Trigger_PLC_Functional_Test_15;
   #Out_Functional_Test.Star_Test_PLC_Functional_Test_15 := #_w1 AND #In_Functional_Test.Star_Test_PLC_Functional_Test_15;
   #Out_Functional_Test.Button_PLC_Functional_Test_15 := #_w1 AND #In_Functional_Test.Button_PLC_Functional_Test_15;
   #Out_Functional_Test.Electrical_Current_Test_Approved_PLC_Functional_Test_15 := #_w1 AND #In_Functional_Test.Electrical_Current_Test_Approved_PLC_Functional_Test_15;
   #Out_Functional_Test.Visual_Test_Approved_PLC_Functional_Test_15 := #_w1 AND #In_Functional_Test.Visual_Test_Approved_PLC_Functional_Test_15;
   IF #_w1 THEN
       #Out_Functional_Test.Electrical_Current_Read_PLC_Functional_Test_15 := #In_Functional_Test.Electrical_Current_Read_PLC_Functional_Test_15;
   END_IF;
   #Out_Functional_Test.Life_Trigger_PLC_Functional_Test_17 := #_w1 AND #In_Functional_Test.Life_Trigger_PLC_Functional_Test_17;
   #Out_Functional_Test.Star_Test_PLC_Functional_Test_17 := #_w1 AND #In_Functional_Test.Star_Test_PLC_Functional_Test_17;
   #Out_Functional_Test.Button_PLC_Functional_Test_17 := #_w1 AND #In_Functional_Test.Button_PLC_Functional_Test_17;
   #Out_Functional_Test.Electrical_Current_Test_Approved_PLC_Functional_Test_17 := #_w1 AND #In_Functional_Test.Electrical_Current_Test_Approved_PLC_Functional_Test_17;
   #Out_Functional_Test.Visual_Test_Approved_PLC_Functional_Test_17 := #_w1 AND #In_Functional_Test.Visual_Test_Approved_PLC_Functional_Test_17;
   IF #_w1 THEN
       #Out_Functional_Test.Electrical_Current_Read_PLC_Functional_Test_17 := #In_Functional_Test.Electrical_Current_Read_PLC_Functional_Test_17;
   END_IF;
   #Out_Functional_Test.Life_Trigger_PLC_Functional_Test_19 := #_w1 AND #In_Functional_Test.Life_Trigger_PLC_Functional_Test_19;
   #Out_Functional_Test.Star_Test_PLC_Functional_Test_19 := #_w1 AND #In_Functional_Test.Star_Test_PLC_Functional_Test_19;
   #Out_Functional_Test.Button_PLC_Functional_Test_19 := #_w1 AND #In_Functional_Test.Button_PLC_Functional_Test_19;
   #Out_Functional_Test.Electrical_Current_Test_Approved_PLC_Functional_Test_19 := #_w1 AND #In_Functional_Test.Electrical_Current_Test_Approved_PLC_Functional_Test_19;
   #Out_Functional_Test.Visual_Test_Approved_PLC_Functional_Test_19 := #_w1 AND #In_Functional_Test.Visual_Test_Approved_PLC_Functional_Test_19;
   IF #_w1 THEN
       #Out_Functional_Test.Electrical_Current_Read_PLC_Functional_Test_19 := #In_Functional_Test.Electrical_Current_Read_PLC_Functional_Test_19;
   END_IF;
   #Out_Functional_Test.Life_Trigger_PLC_Functional_Test_21 := #_w1 AND #In_Functional_Test.Life_Trigger_PLC_Functional_Test_21;
   #Out_Functional_Test.Star_Test_PLC_Functional_Test_21 := #_w1 AND #In_Functional_Test.Star_Test_PLC_Functional_Test_21;
   #Out_Functional_Test.Button_PLC_Functional_Test_21 := #_w1 AND #In_Functional_Test.Button_PLC_Functional_Test_21;
   #Out_Functional_Test.Electrical_Current_Test_Approved_PLC_Functional_Test_21 := #_w1 AND #In_Functional_Test.Electrical_Current_Test_Approved_PLC_Functional_Test_21;
   #Out_Functional_Test.Visual_Test_Approved_PLC_Functional_Test_21 := #_w1 AND #In_Functional_Test.Visual_Test_Approved_PLC_Functional_Test_21;
   IF #_w1 THEN
       #Out_Functional_Test.Electrical_Current_Read_PLC_Functional_Test_21 := #In_Functional_Test.Electrical_Current_Read_PLC_Functional_Test_21;
   END_IF;
   #Out_Functional_Test.Life_Trigger_PLC_Functional_Test_23 := #_w1 AND #In_Functional_Test.Life_Trigger_PLC_Functional_Test_23;
   #Out_Functional_Test.Star_Test_PLC_Functional_Test_23 := #_w1 AND #In_Functional_Test.Star_Test_PLC_Functional_Test_23;
   #Out_Functional_Test.Button_PLC_Functional_Test_23 := #_w1 AND #In_Functional_Test.Button_PLC_Functional_Test_23;
   #Out_Functional_Test.Electrical_Current_Test_Approved_PLC_Functional_Test_23 := #_w1 AND #In_Functional_Test.Electrical_Current_Test_Approved_PLC_Functional_Test_23;
   #Out_Functional_Test.Visual_Test_Approved_PLC_Functional_Test_23 := #_w1 AND #In_Functional_Test.Visual_Test_Approved_PLC_Functional_Test_23;
   IF #_w1 THEN
       #Out_Functional_Test.Electrical_Current_Read_PLC_Functional_Test_23 := #In_Functional_Test.Electrical_Current_Read_PLC_Functional_Test_23;
   END_IF;
   #Out_Functional_Test.Life_Trigger_PLC_Functional_Test_25 := #_w1 AND #In_Functional_Test.Life_Trigger_PLC_Functional_Test_25;
   #Out_Functional_Test.Star_Test_PLC_Functional_Test_25 := #_w1 AND #In_Functional_Test.Star_Test_PLC_Functional_Test_25;
   #Out_Functional_Test.Button_PLC_Functional_Test_25 := #_w1 AND #In_Functional_Test.Button_PLC_Functional_Test_25;
   #Out_Functional_Test.Electrical_Current_Test_Approved_PLC_Functional_Test_25 := #_w1 AND #In_Functional_Test.Electrical_Current_Test_Approved_PLC_Functional_Test_25;
   #Out_Functional_Test.Visual_Test_Approved_PLC_Functional_Test_25 := #_w1 AND #In_Functional_Test.Visual_Test_Approved_PLC_Functional_Test_25;
   IF #_w1 THEN
       #Out_Functional_Test.Electrical_Current_Read_PLC_Functional_Test_25 := #In_Functional_Test.Electrical_Current_Read_PLC_Functional_Test_25;
   END_IF;
   #Out_Functional_Test.Life_Trigger_PLC_Functional_Test_27 := #_w1 AND #In_Functional_Test.Life_Trigger_PLC_Functional_Test_27;
   #Out_Functional_Test.Star_Test_PLC_Functional_Test_27 := #_w1 AND #In_Functional_Test.Star_Test_PLC_Functional_Test_27;
   #Out_Functional_Test.Button_PLC_Functional_Test_27 := #_w1 AND #In_Functional_Test.Button_PLC_Functional_Test_27;
   #Out_Functional_Test.Electrical_Current_Test_Approved_PLC_Functional_Test_27 := #_w1 AND #In_Functional_Test.Electrical_Current_Test_Approved_PLC_Functional_Test_27;
   #Out_Functional_Test.Visual_Test_Approved_PLC_Functional_Test_27 := #_w1 AND #In_Functional_Test.Visual_Test_Approved_PLC_Functional_Test_27;
   IF #_w1 THEN
       #Out_Functional_Test.Electrical_Current_Read_PLC_Functional_Test_27 := #In_Functional_Test.Electrical_Current_Read_PLC_Functional_Test_27;
   END_IF;
   #Out_Functional_Test.Life_Trigger_PLC_Functional_Test_29 := #_w1 AND #In_Functional_Test.Life_Trigger_PLC_Functional_Test_29;
   #Out_Functional_Test.Star_Test_PLC_Functional_Test_29 := #_w1 AND #In_Functional_Test.Star_Test_PLC_Functional_Test_29;
   #Out_Functional_Test.Button_PLC_Functional_Test_29 := #_w1 AND #In_Functional_Test.Button_PLC_Functional_Test_29;
   #Out_Functional_Test.Electrical_Current_Test_Approved_PLC_Functional_Test_29 := #_w1 AND #In_Functional_Test.Electrical_Current_Test_Approved_PLC_Functional_Test_29;
   #Out_Functional_Test.Visual_Test_Approved_PLC_Functional_Test_29 := #_w1 AND #In_Functional_Test.Visual_Test_Approved_PLC_Functional_Test_29;
   IF #_w1 THEN
       #Out_Functional_Test.Electrical_Current_Read_PLC_Functional_Test_29 := #In_Functional_Test.Electrical_Current_Read_PLC_Functional_Test_29;
   END_IF;
END_REGION

REGION Network 7: Functional Test Station 11
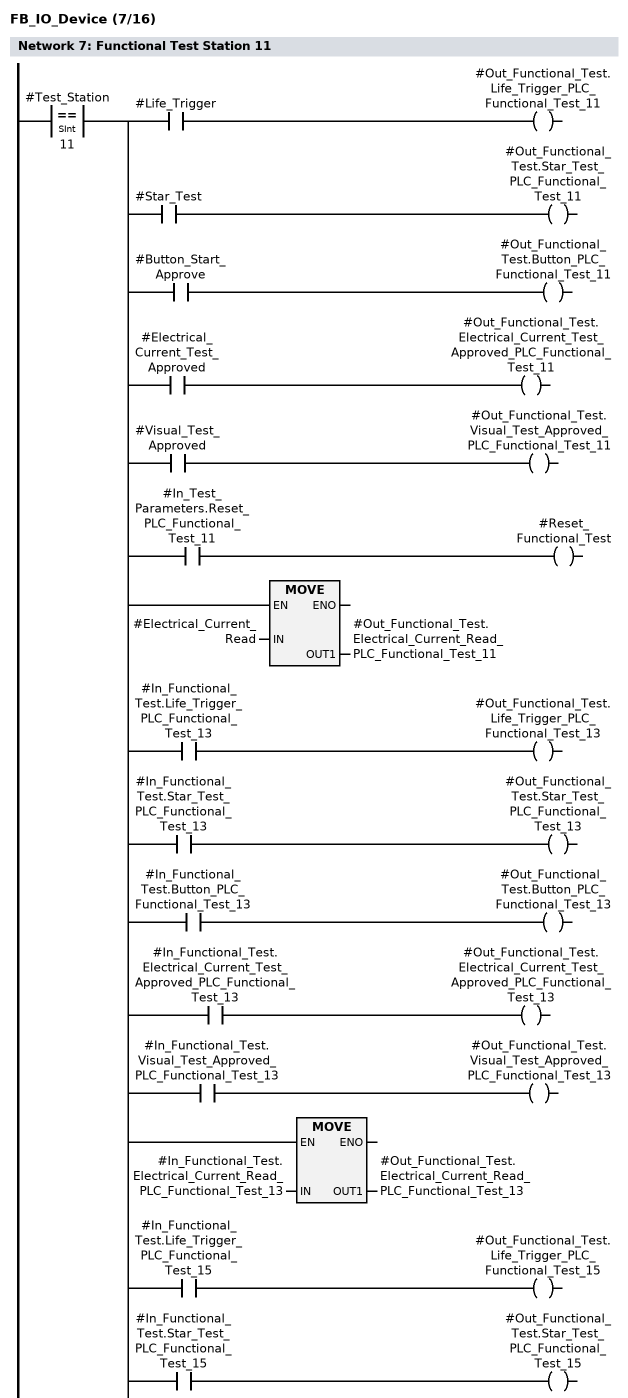
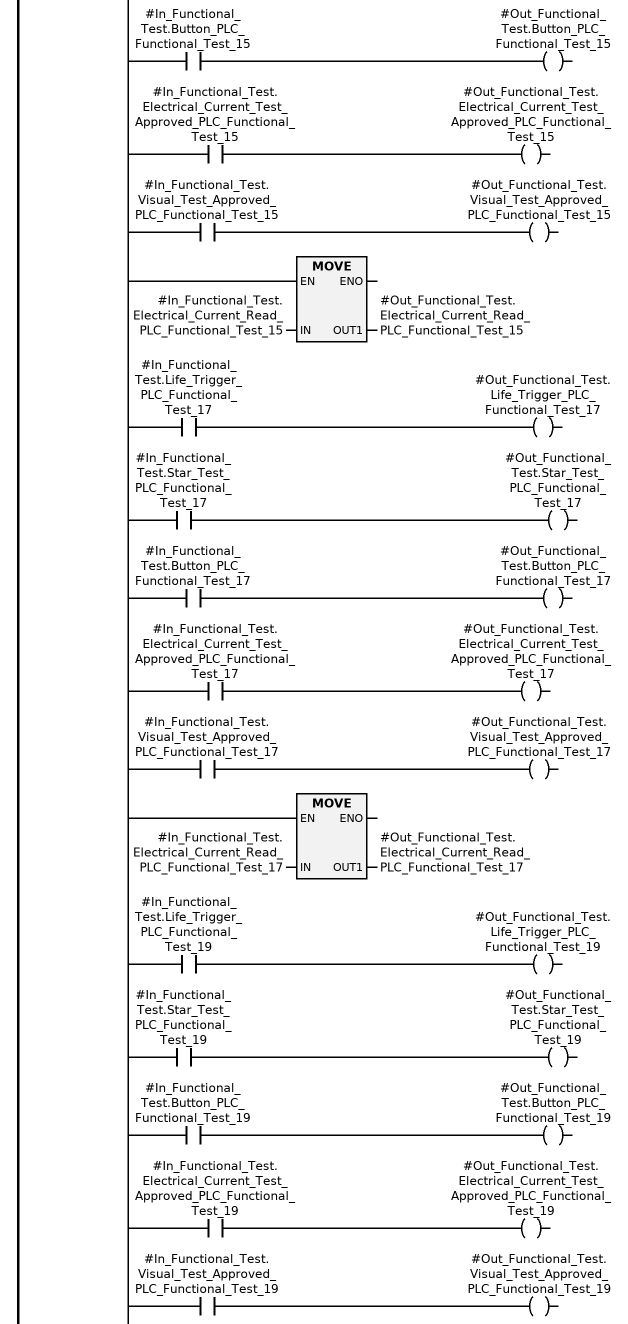
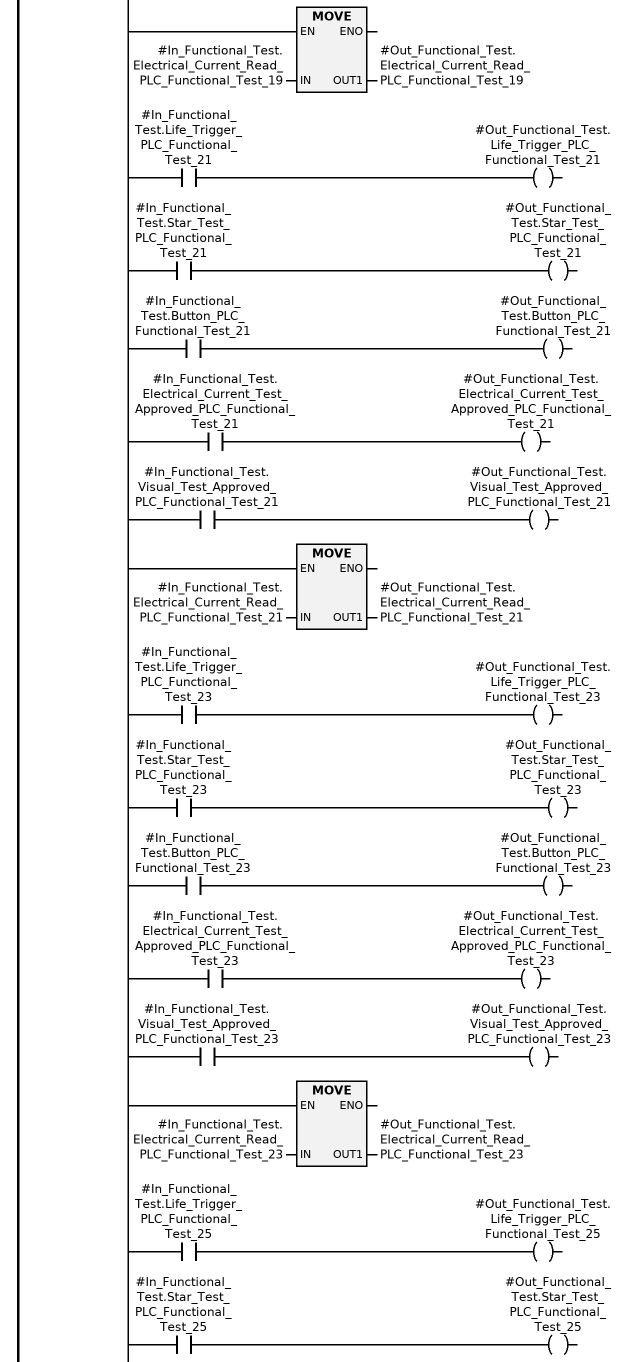
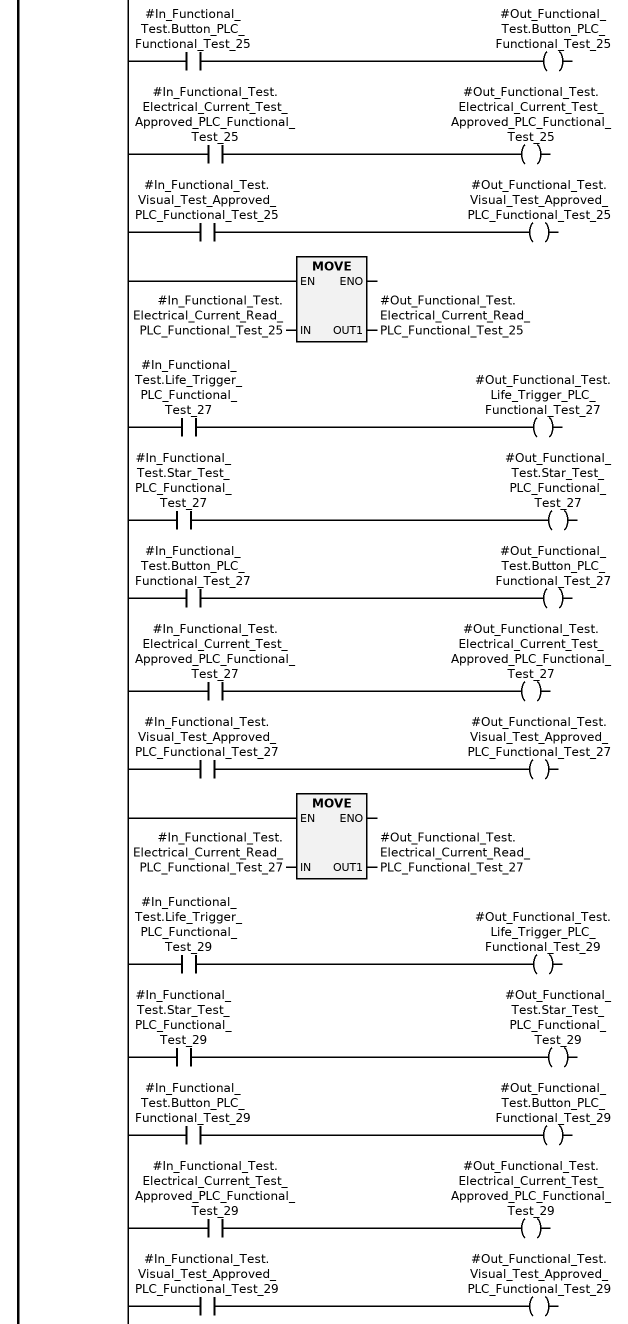
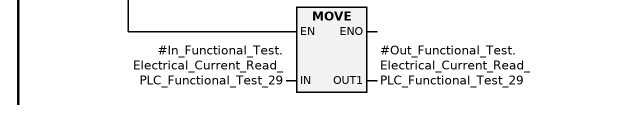
   RUNG wire#powerrail
      { S7_Templates := "SrcType := SInt" } EQ_Contact(in1 := #Test_Station, in2 := 11)
      wire#w1
      Contact( #Life_Trigger )
      Coil( #Out_Functional_Test.Life_Trigger_PLC_Functional_Test_11 )
   END_RUNG
   RUNG wire#w1
      Contact( #Star_Test )
      Coil( #Out_Functional_Test.Star_Test_PLC_Functional_Test_11 )
   END_RUNG
   RUNG wire#w1
      Contact( #Button_Start_Approve )
      Coil( #Out_Functional_Test.Button_PLC_Functional_Test_11 )
   END_RUNG
   RUNG wire#w1
      Contact( #Electrical_Current_Test_Approved )
      Coil( #Out_Functional_Test.Electrical_Current_Test_Approved_PLC_Functional_Test_11 )
   END_RUNG
   RUNG wire#w1
      Contact( #Visual_Test_Approved )
      Coil( #Out_Functional_Test.Visual_Test_Approved_PLC_Functional_Test_11 )
   END_RUNG
   RUNG wire#w1
      Contact( #In_Test_Parameters.Reset_PLC_Functional_Test_11 )
      Coil( #Reset_Functional_Test )
   END_RUNG
   RUNG wire#w1
      Move(in := #Electrical_Current_Read, out1 => #Out_Functional_Test.Electrical_Current_Read_PLC_Functional_Test_11)
   END_RUNG
   RUNG wire#w1
      Contact( #In_Functional_Test.Life_Trigger_PLC_Functional_Test_13 )
      Coil( #Out_Functional_Test.Life_Trigger_PLC_Functional_Test_13 )
   END_RUNG
   RUNG wire#w1
      Contact( #In_Functional_Test.Star_Test_PLC_Functional_Test_13 )
      Coil( #Out_Functional_Test.Star_Test_PLC_Functional_Test_13 )
   END_RUNG
   RUNG wire#w1
      Contact( #In_Functional_Test.Button_PLC_Functional_Test_13 )
      Coil( #Out_Functional_Test.Button_PLC_Functional_Test_13 )
   END_RUNG
   RUNG wire#w1
      Contact( #In_Functional_Test.Electrical_Current_Test_Approved_PLC_Functional_Test_13 )
      Coil( #Out_Functional_Test.Electrical_Current_Test_Approved_PLC_Functional_Test_13 )
   END_RUNG
   RUNG wire#w1
      Contact( #In_Functional_Test.Visual_Test_Approved_PLC_Functional_Test_13 )
      Coil( #Out_Functional_Test.Visual_Test_Approved_PLC_Functional_Test_13 )
   END_RUNG
   RUNG wire#w1
      Move(in := #In_Functional_Test.Electrical_Current_Read_PLC_Functional_Test_13, out1 => #Out_Functional_Test.Electrical_Current_Read_PLC_Functional_Test_13)
   END_RUNG
   RUNG wire#w1
      Contact( #In_Functional_Test.Life_Trigger_PLC_Functional_Test_15 )
      Coil( #Out_Functional_Test.Life_Trigger_PLC_Functional_Test_15 )
   END_RUNG
   RUNG wire#w1
      Contact( #In_Functional_Test.Star_Test_PLC_Functional_Test_15 )
      Coil( #Out_Functional_Test.Star_Test_PLC_Functional_Test_15 )
   END_RUNG
   RUNG wire#w1
      Contact( #In_Functional_Test.Button_PLC_Functional_Test_15 )
      Coil( #Out_Functional_Test.Button_PLC_Functional_Test_15 )
   END_RUNG
   RUNG wire#w1
      Contact( #In_Functional_Test.Electrical_Current_Test_Approved_PLC_Functional_Test_15 )
      Coil( #Out_Functional_Test.Electrical_Current_Test_Approved_PLC_Functional_Test_15 )
   END_RUNG
   RUNG wire#w1
      Contact( #In_Functional_Test.Visual_Test_Approved_PLC_Functional_Test_15 )
      Coil( #Out_Functional_Test.Visual_Test_Approved_PLC_Functional_Test_15 )
   END_RUNG
   RUNG wire#w1
      Move(in := #In_Functional_Test.Electrical_Current_Read_PLC_Functional_Test_15, out1 => #Out_Functional_Test.Electrical_Current_Read_PLC_Functional_Test_15)
   END_RUNG
   RUNG wire#w1
      Contact( #In_Functional_Test.Life_Trigger_PLC_Functional_Test_17 )
      Coil( #Out_Functional_Test.Life_Trigger_PLC_Functional_Test_17 )
   END_RUNG
   RUNG wire#w1
      Contact( #In_Functional_Test.Star_Test_PLC_Functional_Test_17 )
      Coil( #Out_Functional_Test.Star_Test_PLC_Functional_Test_17 )
   END_RUNG
   RUNG wire#w1
      Contact( #In_Functional_Test.Button_PLC_Functional_Test_17 )
      Coil( #Out_Functional_Test.Button_PLC_Functional_Test_17 )
   END_RUNG
   RUNG wire#w1
      Contact( #In_Functional_Test.Electrical_Current_Test_Approved_PLC_Functional_Test_17 )
      Coil( #Out_Functional_Test.Electrical_Current_Test_Approved_PLC_Functional_Test_17 )
   END_RUNG
   RUNG wire#w1
      Contact( #In_Functional_Test.Visual_Test_Approved_PLC_Functional_Test_17 )
      Coil( #Out_Functional_Test.Visual_Test_Approved_PLC_Functional_Test_17 )
   END_RUNG
   RUNG wire#w1
      Move(in := #In_Functional_Test.Electrical_Current_Read_PLC_Functional_Test_17, out1 => #Out_Functional_Test.Electrical_Current_Read_PLC_Functional_Test_17)
   END_RUNG
   RUNG wire#w1
      Contact( #In_Functional_Test.Life_Trigger_PLC_Functional_Test_19 )
      Coil( #Out_Functional_Test.Life_Trigger_PLC_Functional_Test_19 )
   END_RUNG
   RUNG wire#w1
      Contact( #In_Functional_Test.Star_Test_PLC_Functional_Test_19 )
      Coil( #Out_Functional_Test.Star_Test_PLC_Functional_Test_19 )
   END_RUNG
   RUNG wire#w1
      Contact( #In_Functional_Test.Button_PLC_Functional_Test_19 )
      Coil( #Out_Functional_Test.Button_PLC_Functional_Test_19 )
   END_RUNG
   RUNG wire#w1
      Contact( #In_Functional_Test.Electrical_Current_Test_Approved_PLC_Functional_Test_19 )
      Coil( #Out_Functional_Test.Electrical_Current_Test_Approved_PLC_Functional_Test_19 )
   END_RUNG
   RUNG wire#w1
      Contact( #In_Functional_Test.Visual_Test_Approved_PLC_Functional_Test_19 )
      Coil( #Out_Functional_Test.Visual_Test_Approved_PLC_Functional_Test_19 )
   END_RUNG
   RUNG wire#w1
      Move(in := #In_Functional_Test.Electrical_Current_Read_PLC_Functional_Test_19, out1 => #Out_Functional_Test.Electrical_Current_Read_PLC_Functional_Test_19)
   END_RUNG
   RUNG wire#w1
      Contact( #In_Functional_Test.Life_Trigger_PLC_Functional_Test_21 )
      Coil( #Out_Functional_Test.Life_Trigger_PLC_Functional_Test_21 )
   END_RUNG
   RUNG wire#w1
      Contact( #In_Functional_Test.Star_Test_PLC_Functional_Test_21 )
      Coil( #Out_Functional_Test.Star_Test_PLC_Functional_Test_21 )
   END_RUNG
   RUNG wire#w1
      Contact( #In_Functional_Test.Button_PLC_Functional_Test_21 )
      Coil( #Out_Functional_Test.Button_PLC_Functional_Test_21 )
   END_RUNG
   RUNG wire#w1
      Contact( #In_Functional_Test.Electrical_Current_Test_Approved_PLC_Functional_Test_21 )
      Coil( #Out_Functional_Test.Electrical_Current_Test_Approved_PLC_Functional_Test_21 )
   END_RUNG
   RUNG wire#w1
      Contact( #In_Functional_Test.Visual_Test_Approved_PLC_Functional_Test_21 )
      Coil( #Out_Functional_Test.Visual_Test_Approved_PLC_Functional_Test_21 )
   END_RUNG
   RUNG wire#w1
      Move(in := #In_Functional_Test.Electrical_Current_Read_PLC_Functional_Test_21, out1 => #Out_Functional_Test.Electrical_Current_Read_PLC_Functional_Test_21)
   END_RUNG
   RUNG wire#w1
      Contact( #In_Functional_Test.Life_Trigger_PLC_Functional_Test_23 )
      Coil( #Out_Functional_Test.Life_Trigger_PLC_Functional_Test_23 )
   END_RUNG
   RUNG wire#w1
      Contact( #In_Functional_Test.Star_Test_PLC_Functional_Test_23 )
      Coil( #Out_Functional_Test.Star_Test_PLC_Functional_Test_23 )
   END_RUNG
   RUNG wire#w1
      Contact( #In_Functional_Test.Button_PLC_Functional_Test_23 )
      Coil( #Out_Functional_Test.Button_PLC_Functional_Test_23 )
   END_RUNG
   RUNG wire#w1
      Contact( #In_Functional_Test.Electrical_Current_Test_Approved_PLC_Functional_Test_23 )
      Coil( #Out_Functional_Test.Electrical_Current_Test_Approved_PLC_Functional_Test_23 )
   END_RUNG
   RUNG wire#w1
      Contact( #In_Functional_Test.Visual_Test_Approved_PLC_Functional_Test_23 )
      Coil( #Out_Functional_Test.Visual_Test_Approved_PLC_Functional_Test_23 )
   END_RUNG
   RUNG wire#w1
      Move(in := #In_Functional_Test.Electrical_Current_Read_PLC_Functional_Test_23, out1 => #Out_Functional_Test.Electrical_Current_Read_PLC_Functional_Test_23)
   END_RUNG
   RUNG wire#w1
      Contact( #In_Functional_Test.Life_Trigger_PLC_Functional_Test_25 )
      Coil( #Out_Functional_Test.Life_Trigger_PLC_Functional_Test_25 )
   END_RUNG
   RUNG wire#w1
      Contact( #In_Functional_Test.Star_Test_PLC_Functional_Test_25 )
      Coil( #Out_Functional_Test.Star_Test_PLC_Functional_Test_25 )
   END_RUNG
   RUNG wire#w1
      Contact( #In_Functional_Test.Button_PLC_Functional_Test_25 )
      Coil( #Out_Functional_Test.Button_PLC_Functional_Test_25 )
   END_RUNG
   RUNG wire#w1
      Contact( #In_Functional_Test.Electrical_Current_Test_Approved_PLC_Functional_Test_25 )
      Coil( #Out_Functional_Test.Electrical_Current_Test_Approved_PLC_Functional_Test_25 )
   END_RUNG
   RUNG wire#w1
      Contact( #In_Functional_Test.Visual_Test_Approved_PLC_Functional_Test_25 )
      Coil( #Out_Functional_Test.Visual_Test_Approved_PLC_Functional_Test_25 )
   END_RUNG
   RUNG wire#w1
      Move(in := #In_Functional_Test.Electrical_Current_Read_PLC_Functional_Test_25, out1 => #Out_Functional_Test.Electrical_Current_Read_PLC_Functional_Test_25)
   END_RUNG
   RUNG wire#w1
      Contact( #In_Functional_Test.Life_Trigger_PLC_Functional_Test_27 )
      Coil( #Out_Functional_Test.Life_Trigger_PLC_Functional_Test_27 )
   END_RUNG
   RUNG wire#w1
      Contact( #In_Functional_Test.Star_Test_PLC_Functional_Test_27 )
      Coil( #Out_Functional_Test.Star_Test_PLC_Functional_Test_27 )
   END_RUNG
   RUNG wire#w1
      Contact( #In_Functional_Test.Button_PLC_Functional_Test_27 )
      Coil( #Out_Functional_Test.Button_PLC_Functional_Test_27 )
   END_RUNG
   RUNG wire#w1
      Contact( #In_Functional_Test.Electrical_Current_Test_Approved_PLC_Functional_Test_27 )
      Coil( #Out_Functional_Test.Electrical_Current_Test_Approved_PLC_Functional_Test_27 )
   END_RUNG
   RUNG wire#w1
      Contact( #In_Functional_Test.Visual_Test_Approved_PLC_Functional_Test_27 )
      Coil( #Out_Functional_Test.Visual_Test_Approved_PLC_Functional_Test_27 )
   END_RUNG
   RUNG wire#w1
      Move(in := #In_Functional_Test.Electrical_Current_Read_PLC_Functional_Test_27, out1 => #Out_Functional_Test.Electrical_Current_Read_PLC_Functional_Test_27)
   END_RUNG
   RUNG wire#w1
      Contact( #In_Functional_Test.Life_Trigger_PLC_Functional_Test_29 )
      Coil( #Out_Functional_Test.Life_Trigger_PLC_Functional_Test_29 )
   END_RUNG
   RUNG wire#w1
      Contact( #In_Functional_Test.Star_Test_PLC_Functional_Test_29 )
      Coil( #Out_Functional_Test.Star_Test_PLC_Functional_Test_29 )
   END_RUNG
   RUNG wire#w1
      Contact( #In_Functional_Test.Button_PLC_Functional_Test_29 )
      Coil( #Out_Functional_Test.Button_PLC_Functional_Test_29 )
   END_RUNG
   RUNG wire#w1
      Contact( #In_Functional_Test.Electrical_Current_Test_Approved_PLC_Functional_Test_29 )
      Coil( #Out_Functional_Test.Electrical_Current_Test_Approved_PLC_Functional_Test_29 )
   END_RUNG
   RUNG wire#w1
      Contact( #In_Functional_Test.Visual_Test_Approved_PLC_Functional_Test_29 )
      Coil( #Out_Functional_Test.Visual_Test_Approved_PLC_Functional_Test_29 )
   END_RUNG
   RUNG wire#w1
      Move(in := #In_Functional_Test.Electrical_Current_Read_PLC_Functional_Test_29, out1 => #Out_Functional_Test.Electrical_Current_Read_PLC_Functional_Test_29)
   END_RUNG
   // the same network as SCL:
   #_w1 := #Test_Station = 11;
   #Out_Functional_Test.Life_Trigger_PLC_Functional_Test_11 := #_w1 AND #Life_Trigger;
   #Out_Functional_Test.Star_Test_PLC_Functional_Test_11 := #_w1 AND #Star_Test;
   #Out_Functional_Test.Button_PLC_Functional_Test_11 := #_w1 AND #Button_Start_Approve;
   #Out_Functional_Test.Electrical_Current_Test_Approved_PLC_Functional_Test_11 := #_w1 AND #Electrical_Current_Test_Approved;
   #Out_Functional_Test.Visual_Test_Approved_PLC_Functional_Test_11 := #_w1 AND #Visual_Test_Approved;
   #Reset_Functional_Test := #_w1 AND #In_Test_Parameters.Reset_PLC_Functional_Test_11;
   IF #_w1 THEN
       #Out_Functional_Test.Electrical_Current_Read_PLC_Functional_Test_11 := #Electrical_Current_Read;
   END_IF;
   #Out_Functional_Test.Life_Trigger_PLC_Functional_Test_13 := #_w1 AND #In_Functional_Test.Life_Trigger_PLC_Functional_Test_13;
   #Out_Functional_Test.Star_Test_PLC_Functional_Test_13 := #_w1 AND #In_Functional_Test.Star_Test_PLC_Functional_Test_13;
   #Out_Functional_Test.Button_PLC_Functional_Test_13 := #_w1 AND #In_Functional_Test.Button_PLC_Functional_Test_13;
   #Out_Functional_Test.Electrical_Current_Test_Approved_PLC_Functional_Test_13 := #_w1 AND #In_Functional_Test.Electrical_Current_Test_Approved_PLC_Functional_Test_13;
   #Out_Functional_Test.Visual_Test_Approved_PLC_Functional_Test_13 := #_w1 AND #In_Functional_Test.Visual_Test_Approved_PLC_Functional_Test_13;
   IF #_w1 THEN
       #Out_Functional_Test.Electrical_Current_Read_PLC_Functional_Test_13 := #In_Functional_Test.Electrical_Current_Read_PLC_Functional_Test_13;
   END_IF;
   #Out_Functional_Test.Life_Trigger_PLC_Functional_Test_15 := #_w1 AND #In_Functional_Test.Life_Trigger_PLC_Functional_Test_15;
   #Out_Functional_Test.Star_Test_PLC_Functional_Test_15 := #_w1 AND #In_Functional_Test.Star_Test_PLC_Functional_Test_15;
   #Out_Functional_Test.Button_PLC_Functional_Test_15 := #_w1 AND #In_Functional_Test.Button_PLC_Functional_Test_15;
   #Out_Functional_Test.Electrical_Current_Test_Approved_PLC_Functional_Test_15 := #_w1 AND #In_Functional_Test.Electrical_Current_Test_Approved_PLC_Functional_Test_15;
   #Out_Functional_Test.Visual_Test_Approved_PLC_Functional_Test_15 := #_w1 AND #In_Functional_Test.Visual_Test_Approved_PLC_Functional_Test_15;
   IF #_w1 THEN
       #Out_Functional_Test.Electrical_Current_Read_PLC_Functional_Test_15 := #In_Functional_Test.Electrical_Current_Read_PLC_Functional_Test_15;
   END_IF;
   #Out_Functional_Test.Life_Trigger_PLC_Functional_Test_17 := #_w1 AND #In_Functional_Test.Life_Trigger_PLC_Functional_Test_17;
   #Out_Functional_Test.Star_Test_PLC_Functional_Test_17 := #_w1 AND #In_Functional_Test.Star_Test_PLC_Functional_Test_17;
   #Out_Functional_Test.Button_PLC_Functional_Test_17 := #_w1 AND #In_Functional_Test.Button_PLC_Functional_Test_17;
   #Out_Functional_Test.Electrical_Current_Test_Approved_PLC_Functional_Test_17 := #_w1 AND #In_Functional_Test.Electrical_Current_Test_Approved_PLC_Functional_Test_17;
   #Out_Functional_Test.Visual_Test_Approved_PLC_Functional_Test_17 := #_w1 AND #In_Functional_Test.Visual_Test_Approved_PLC_Functional_Test_17;
   IF #_w1 THEN
       #Out_Functional_Test.Electrical_Current_Read_PLC_Functional_Test_17 := #In_Functional_Test.Electrical_Current_Read_PLC_Functional_Test_17;
   END_IF;
   #Out_Functional_Test.Life_Trigger_PLC_Functional_Test_19 := #_w1 AND #In_Functional_Test.Life_Trigger_PLC_Functional_Test_19;
   #Out_Functional_Test.Star_Test_PLC_Functional_Test_19 := #_w1 AND #In_Functional_Test.Star_Test_PLC_Functional_Test_19;
   #Out_Functional_Test.Button_PLC_Functional_Test_19 := #_w1 AND #In_Functional_Test.Button_PLC_Functional_Test_19;
   #Out_Functional_Test.Electrical_Current_Test_Approved_PLC_Functional_Test_19 := #_w1 AND #In_Functional_Test.Electrical_Current_Test_Approved_PLC_Functional_Test_19;
   #Out_Functional_Test.Visual_Test_Approved_PLC_Functional_Test_19 := #_w1 AND #In_Functional_Test.Visual_Test_Approved_PLC_Functional_Test_19;
   IF #_w1 THEN
       #Out_Functional_Test.Electrical_Current_Read_PLC_Functional_Test_19 := #In_Functional_Test.Electrical_Current_Read_PLC_Functional_Test_19;
   END_IF;
   #Out_Functional_Test.Life_Trigger_PLC_Functional_Test_21 := #_w1 AND #In_Functional_Test.Life_Trigger_PLC_Functional_Test_21;
   #Out_Functional_Test.Star_Test_PLC_Functional_Test_21 := #_w1 AND #In_Functional_Test.Star_Test_PLC_Functional_Test_21;
   #Out_Functional_Test.Button_PLC_Functional_Test_21 := #_w1 AND #In_Functional_Test.Button_PLC_Functional_Test_21;
   #Out_Functional_Test.Electrical_Current_Test_Approved_PLC_Functional_Test_21 := #_w1 AND #In_Functional_Test.Electrical_Current_Test_Approved_PLC_Functional_Test_21;
   #Out_Functional_Test.Visual_Test_Approved_PLC_Functional_Test_21 := #_w1 AND #In_Functional_Test.Visual_Test_Approved_PLC_Functional_Test_21;
   IF #_w1 THEN
       #Out_Functional_Test.Electrical_Current_Read_PLC_Functional_Test_21 := #In_Functional_Test.Electrical_Current_Read_PLC_Functional_Test_21;
   END_IF;
   #Out_Functional_Test.Life_Trigger_PLC_Functional_Test_23 := #_w1 AND #In_Functional_Test.Life_Trigger_PLC_Functional_Test_23;
   #Out_Functional_Test.Star_Test_PLC_Functional_Test_23 := #_w1 AND #In_Functional_Test.Star_Test_PLC_Functional_Test_23;
   #Out_Functional_Test.Button_PLC_Functional_Test_23 := #_w1 AND #In_Functional_Test.Button_PLC_Functional_Test_23;
   #Out_Functional_Test.Electrical_Current_Test_Approved_PLC_Functional_Test_23 := #_w1 AND #In_Functional_Test.Electrical_Current_Test_Approved_PLC_Functional_Test_23;
   #Out_Functional_Test.Visual_Test_Approved_PLC_Functional_Test_23 := #_w1 AND #In_Functional_Test.Visual_Test_Approved_PLC_Functional_Test_23;
   IF #_w1 THEN
       #Out_Functional_Test.Electrical_Current_Read_PLC_Functional_Test_23 := #In_Functional_Test.Electrical_Current_Read_PLC_Functional_Test_23;
   END_IF;
   #Out_Functional_Test.Life_Trigger_PLC_Functional_Test_25 := #_w1 AND #In_Functional_Test.Life_Trigger_PLC_Functional_Test_25;
   #Out_Functional_Test.Star_Test_PLC_Functional_Test_25 := #_w1 AND #In_Functional_Test.Star_Test_PLC_Functional_Test_25;
   #Out_Functional_Test.Button_PLC_Functional_Test_25 := #_w1 AND #In_Functional_Test.Button_PLC_Functional_Test_25;
   #Out_Functional_Test.Electrical_Current_Test_Approved_PLC_Functional_Test_25 := #_w1 AND #In_Functional_Test.Electrical_Current_Test_Approved_PLC_Functional_Test_25;
   #Out_Functional_Test.Visual_Test_Approved_PLC_Functional_Test_25 := #_w1 AND #In_Functional_Test.Visual_Test_Approved_PLC_Functional_Test_25;
   IF #_w1 THEN
       #Out_Functional_Test.Electrical_Current_Read_PLC_Functional_Test_25 := #In_Functional_Test.Electrical_Current_Read_PLC_Functional_Test_25;
   END_IF;
   #Out_Functional_Test.Life_Trigger_PLC_Functional_Test_27 := #_w1 AND #In_Functional_Test.Life_Trigger_PLC_Functional_Test_27;
   #Out_Functional_Test.Star_Test_PLC_Functional_Test_27 := #_w1 AND #In_Functional_Test.Star_Test_PLC_Functional_Test_27;
   #Out_Functional_Test.Button_PLC_Functional_Test_27 := #_w1 AND #In_Functional_Test.Button_PLC_Functional_Test_27;
   #Out_Functional_Test.Electrical_Current_Test_Approved_PLC_Functional_Test_27 := #_w1 AND #In_Functional_Test.Electrical_Current_Test_Approved_PLC_Functional_Test_27;
   #Out_Functional_Test.Visual_Test_Approved_PLC_Functional_Test_27 := #_w1 AND #In_Functional_Test.Visual_Test_Approved_PLC_Functional_Test_27;
   IF #_w1 THEN
       #Out_Functional_Test.Electrical_Current_Read_PLC_Functional_Test_27 := #In_Functional_Test.Electrical_Current_Read_PLC_Functional_Test_27;
   END_IF;
   #Out_Functional_Test.Life_Trigger_PLC_Functional_Test_29 := #_w1 AND #In_Functional_Test.Life_Trigger_PLC_Functional_Test_29;
   #Out_Functional_Test.Star_Test_PLC_Functional_Test_29 := #_w1 AND #In_Functional_Test.Star_Test_PLC_Functional_Test_29;
   #Out_Functional_Test.Button_PLC_Functional_Test_29 := #_w1 AND #In_Functional_Test.Button_PLC_Functional_Test_29;
   #Out_Functional_Test.Electrical_Current_Test_Approved_PLC_Functional_Test_29 := #_w1 AND #In_Functional_Test.Electrical_Current_Test_Approved_PLC_Functional_Test_29;
   #Out_Functional_Test.Visual_Test_Approved_PLC_Functional_Test_29 := #_w1 AND #In_Functional_Test.Visual_Test_Approved_PLC_Functional_Test_29;
   IF #_w1 THEN
       #Out_Functional_Test.Electrical_Current_Read_PLC_Functional_Test_29 := #In_Functional_Test.Electrical_Current_Read_PLC_Functional_Test_29;
   END_IF;
END_REGION

REGION Network 8: Functional Test Station 13
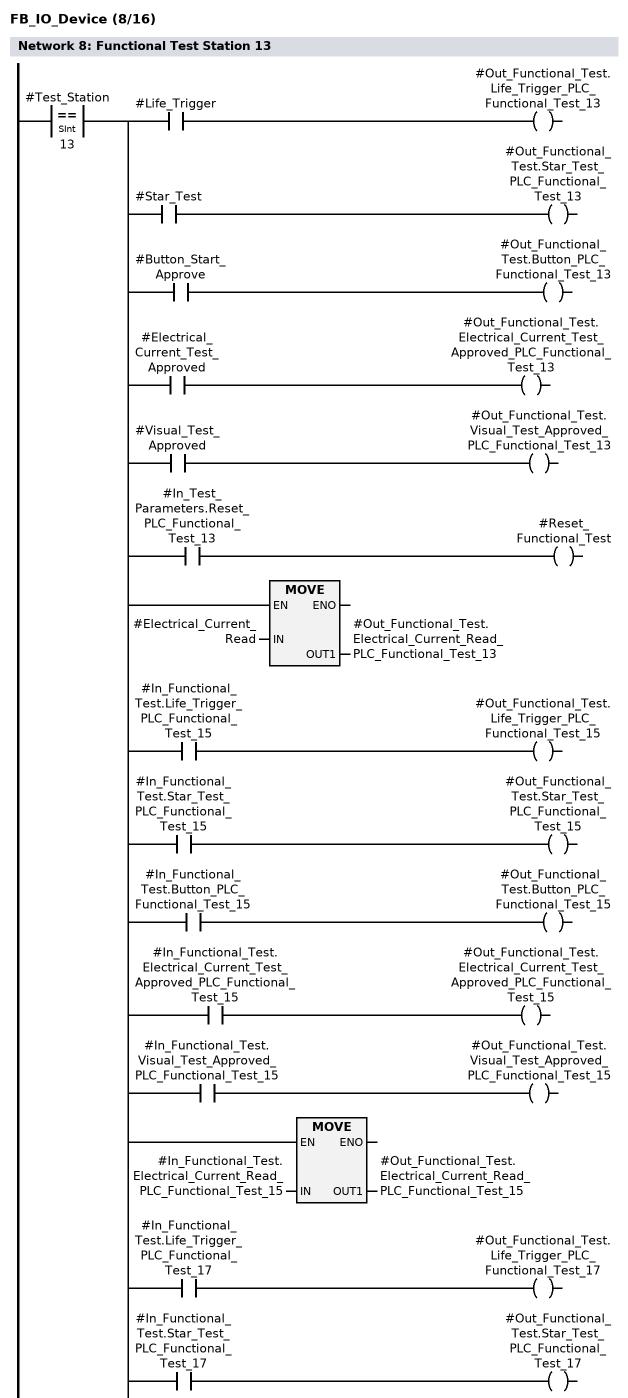
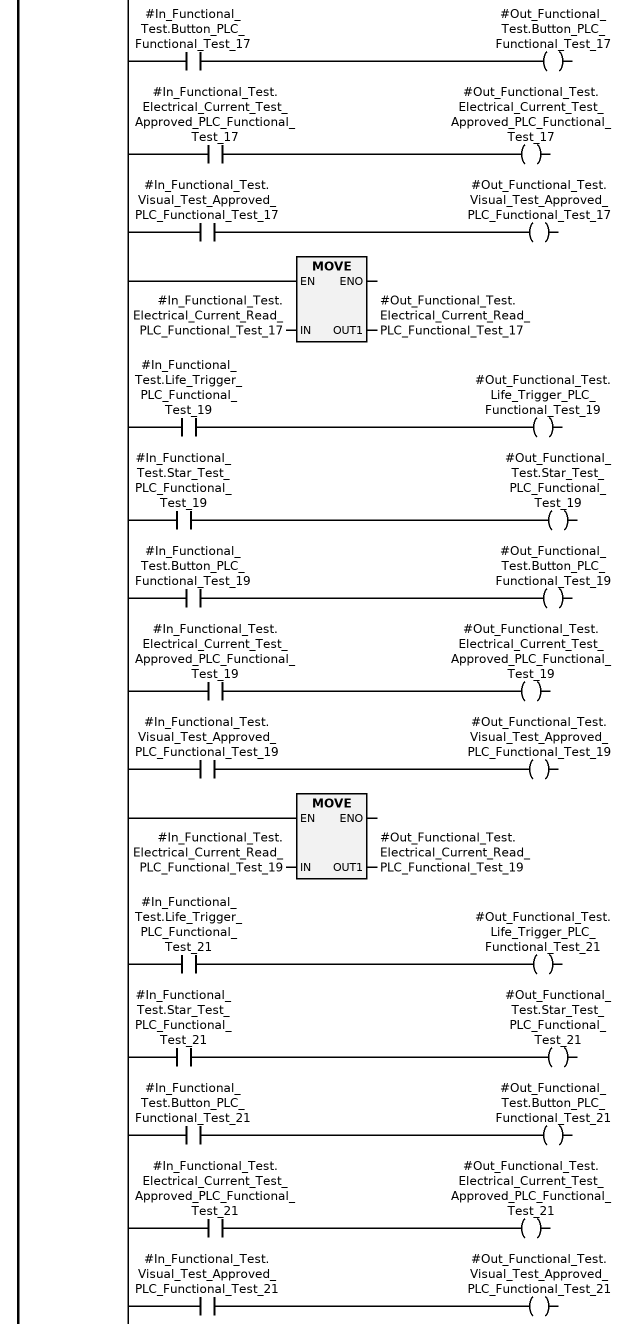
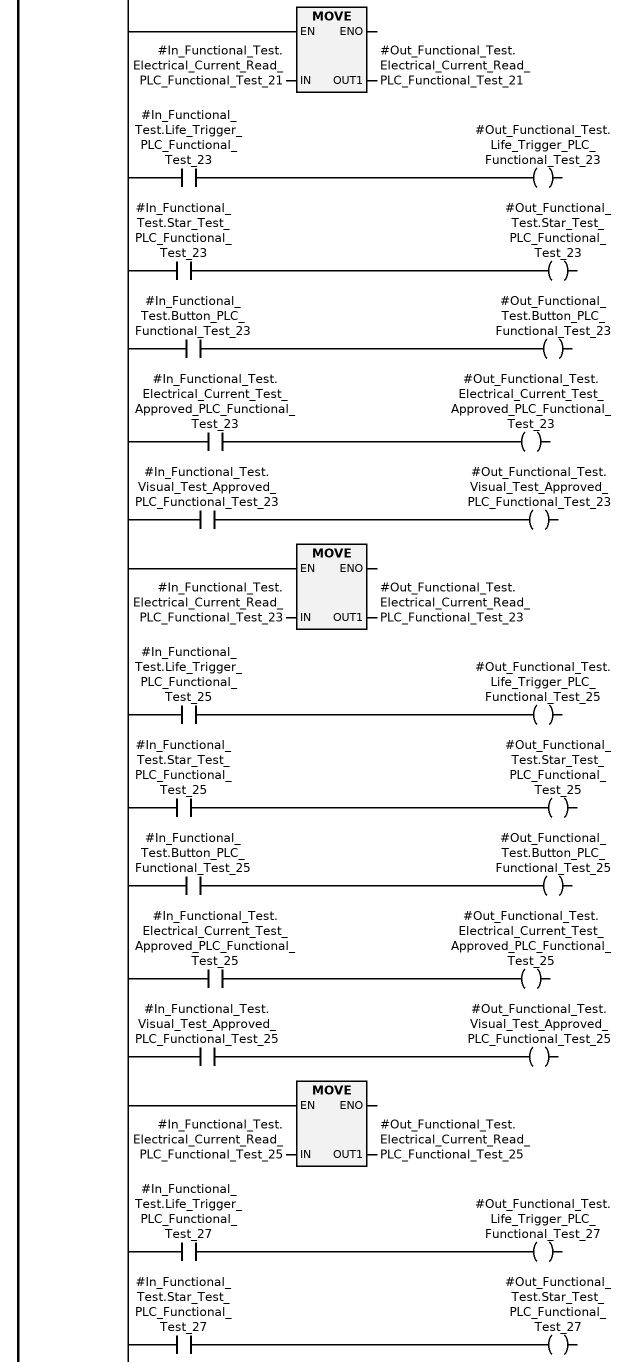
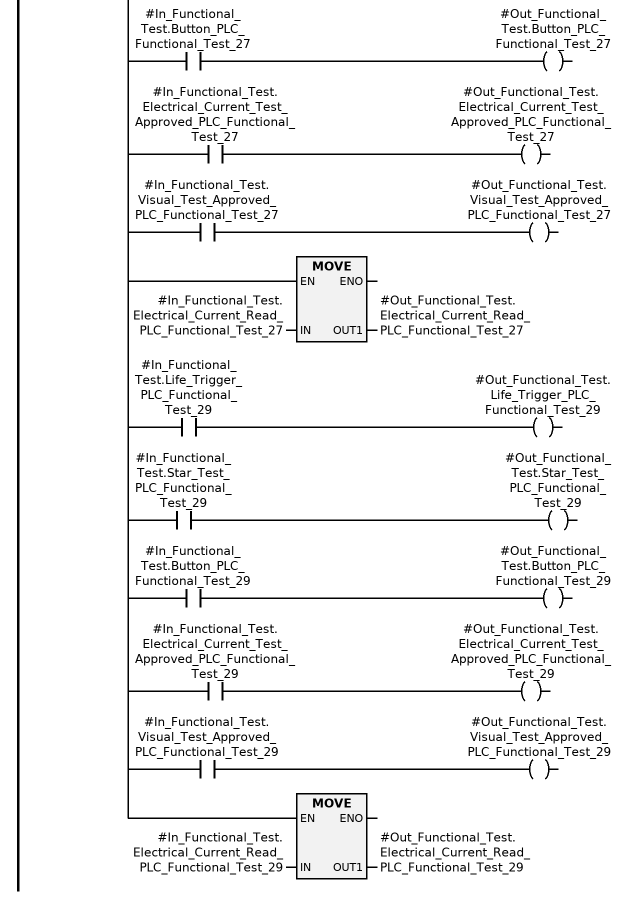
   RUNG wire#powerrail
      { S7_Templates := "SrcType := SInt" } EQ_Contact(in1 := #Test_Station, in2 := 13)
      wire#w1
      Contact( #Life_Trigger )
      Coil( #Out_Functional_Test.Life_Trigger_PLC_Functional_Test_13 )
   END_RUNG
   RUNG wire#w1
      Contact( #Star_Test )
      Coil( #Out_Functional_Test.Star_Test_PLC_Functional_Test_13 )
   END_RUNG
   RUNG wire#w1
      Contact( #Button_Start_Approve )
      Coil( #Out_Functional_Test.Button_PLC_Functional_Test_13 )
   END_RUNG
   RUNG wire#w1
      Contact( #Electrical_Current_Test_Approved )
      Coil( #Out_Functional_Test.Electrical_Current_Test_Approved_PLC_Functional_Test_13 )
   END_RUNG
   RUNG wire#w1
      Contact( #Visual_Test_Approved )
      Coil( #Out_Functional_Test.Visual_Test_Approved_PLC_Functional_Test_13 )
   END_RUNG
   RUNG wire#w1
      Contact( #In_Test_Parameters.Reset_PLC_Functional_Test_13 )
      Coil( #Reset_Functional_Test )
   END_RUNG
   RUNG wire#w1
      Move(in := #Electrical_Current_Read, out1 => #Out_Functional_Test.Electrical_Current_Read_PLC_Functional_Test_13)
   END_RUNG
   RUNG wire#w1
      Contact( #In_Functional_Test.Life_Trigger_PLC_Functional_Test_15 )
      Coil( #Out_Functional_Test.Life_Trigger_PLC_Functional_Test_15 )
   END_RUNG
   RUNG wire#w1
      Contact( #In_Functional_Test.Star_Test_PLC_Functional_Test_15 )
      Coil( #Out_Functional_Test.Star_Test_PLC_Functional_Test_15 )
   END_RUNG
   RUNG wire#w1
      Contact( #In_Functional_Test.Button_PLC_Functional_Test_15 )
      Coil( #Out_Functional_Test.Button_PLC_Functional_Test_15 )
   END_RUNG
   RUNG wire#w1
      Contact( #In_Functional_Test.Electrical_Current_Test_Approved_PLC_Functional_Test_15 )
      Coil( #Out_Functional_Test.Electrical_Current_Test_Approved_PLC_Functional_Test_15 )
   END_RUNG
   RUNG wire#w1
      Contact( #In_Functional_Test.Visual_Test_Approved_PLC_Functional_Test_15 )
      Coil( #Out_Functional_Test.Visual_Test_Approved_PLC_Functional_Test_15 )
   END_RUNG
   RUNG wire#w1
      Move(in := #In_Functional_Test.Electrical_Current_Read_PLC_Functional_Test_15, out1 => #Out_Functional_Test.Electrical_Current_Read_PLC_Functional_Test_15)
   END_RUNG
   RUNG wire#w1
      Contact( #In_Functional_Test.Life_Trigger_PLC_Functional_Test_17 )
      Coil( #Out_Functional_Test.Life_Trigger_PLC_Functional_Test_17 )
   END_RUNG
   RUNG wire#w1
      Contact( #In_Functional_Test.Star_Test_PLC_Functional_Test_17 )
      Coil( #Out_Functional_Test.Star_Test_PLC_Functional_Test_17 )
   END_RUNG
   RUNG wire#w1
      Contact( #In_Functional_Test.Button_PLC_Functional_Test_17 )
      Coil( #Out_Functional_Test.Button_PLC_Functional_Test_17 )
   END_RUNG
   RUNG wire#w1
      Contact( #In_Functional_Test.Electrical_Current_Test_Approved_PLC_Functional_Test_17 )
      Coil( #Out_Functional_Test.Electrical_Current_Test_Approved_PLC_Functional_Test_17 )
   END_RUNG
   RUNG wire#w1
      Contact( #In_Functional_Test.Visual_Test_Approved_PLC_Functional_Test_17 )
      Coil( #Out_Functional_Test.Visual_Test_Approved_PLC_Functional_Test_17 )
   END_RUNG
   RUNG wire#w1
      Move(in := #In_Functional_Test.Electrical_Current_Read_PLC_Functional_Test_17, out1 => #Out_Functional_Test.Electrical_Current_Read_PLC_Functional_Test_17)
   END_RUNG
   RUNG wire#w1
      Contact( #In_Functional_Test.Life_Trigger_PLC_Functional_Test_19 )
      Coil( #Out_Functional_Test.Life_Trigger_PLC_Functional_Test_19 )
   END_RUNG
   RUNG wire#w1
      Contact( #In_Functional_Test.Star_Test_PLC_Functional_Test_19 )
      Coil( #Out_Functional_Test.Star_Test_PLC_Functional_Test_19 )
   END_RUNG
   RUNG wire#w1
      Contact( #In_Functional_Test.Button_PLC_Functional_Test_19 )
      Coil( #Out_Functional_Test.Button_PLC_Functional_Test_19 )
   END_RUNG
   RUNG wire#w1
      Contact( #In_Functional_Test.Electrical_Current_Test_Approved_PLC_Functional_Test_19 )
      Coil( #Out_Functional_Test.Electrical_Current_Test_Approved_PLC_Functional_Test_19 )
   END_RUNG
   RUNG wire#w1
      Contact( #In_Functional_Test.Visual_Test_Approved_PLC_Functional_Test_19 )
      Coil( #Out_Functional_Test.Visual_Test_Approved_PLC_Functional_Test_19 )
   END_RUNG
   RUNG wire#w1
      Move(in := #In_Functional_Test.Electrical_Current_Read_PLC_Functional_Test_19, out1 => #Out_Functional_Test.Electrical_Current_Read_PLC_Functional_Test_19)
   END_RUNG
   RUNG wire#w1
      Contact( #In_Functional_Test.Life_Trigger_PLC_Functional_Test_21 )
      Coil( #Out_Functional_Test.Life_Trigger_PLC_Functional_Test_21 )
   END_RUNG
   RUNG wire#w1
      Contact( #In_Functional_Test.Star_Test_PLC_Functional_Test_21 )
      Coil( #Out_Functional_Test.Star_Test_PLC_Functional_Test_21 )
   END_RUNG
   RUNG wire#w1
      Contact( #In_Functional_Test.Button_PLC_Functional_Test_21 )
      Coil( #Out_Functional_Test.Button_PLC_Functional_Test_21 )
   END_RUNG
   RUNG wire#w1
      Contact( #In_Functional_Test.Electrical_Current_Test_Approved_PLC_Functional_Test_21 )
      Coil( #Out_Functional_Test.Electrical_Current_Test_Approved_PLC_Functional_Test_21 )
   END_RUNG
   RUNG wire#w1
      Contact( #In_Functional_Test.Visual_Test_Approved_PLC_Functional_Test_21 )
      Coil( #Out_Functional_Test.Visual_Test_Approved_PLC_Functional_Test_21 )
   END_RUNG
   RUNG wire#w1
      Move(in := #In_Functional_Test.Electrical_Current_Read_PLC_Functional_Test_21, out1 => #Out_Functional_Test.Electrical_Current_Read_PLC_Functional_Test_21)
   END_RUNG
   RUNG wire#w1
      Contact( #In_Functional_Test.Life_Trigger_PLC_Functional_Test_23 )
      Coil( #Out_Functional_Test.Life_Trigger_PLC_Functional_Test_23 )
   END_RUNG
   RUNG wire#w1
      Contact( #In_Functional_Test.Star_Test_PLC_Functional_Test_23 )
      Coil( #Out_Functional_Test.Star_Test_PLC_Functional_Test_23 )
   END_RUNG
   RUNG wire#w1
      Contact( #In_Functional_Test.Button_PLC_Functional_Test_23 )
      Coil( #Out_Functional_Test.Button_PLC_Functional_Test_23 )
   END_RUNG
   RUNG wire#w1
      Contact( #In_Functional_Test.Electrical_Current_Test_Approved_PLC_Functional_Test_23 )
      Coil( #Out_Functional_Test.Electrical_Current_Test_Approved_PLC_Functional_Test_23 )
   END_RUNG
   RUNG wire#w1
      Contact( #In_Functional_Test.Visual_Test_Approved_PLC_Functional_Test_23 )
      Coil( #Out_Functional_Test.Visual_Test_Approved_PLC_Functional_Test_23 )
   END_RUNG
   RUNG wire#w1
      Move(in := #In_Functional_Test.Electrical_Current_Read_PLC_Functional_Test_23, out1 => #Out_Functional_Test.Electrical_Current_Read_PLC_Functional_Test_23)
   END_RUNG
   RUNG wire#w1
      Contact( #In_Functional_Test.Life_Trigger_PLC_Functional_Test_25 )
      Coil( #Out_Functional_Test.Life_Trigger_PLC_Functional_Test_25 )
   END_RUNG
   RUNG wire#w1
      Contact( #In_Functional_Test.Star_Test_PLC_Functional_Test_25 )
      Coil( #Out_Functional_Test.Star_Test_PLC_Functional_Test_25 )
   END_RUNG
   RUNG wire#w1
      Contact( #In_Functional_Test.Button_PLC_Functional_Test_25 )
      Coil( #Out_Functional_Test.Button_PLC_Functional_Test_25 )
   END_RUNG
   RUNG wire#w1
      Contact( #In_Functional_Test.Electrical_Current_Test_Approved_PLC_Functional_Test_25 )
      Coil( #Out_Functional_Test.Electrical_Current_Test_Approved_PLC_Functional_Test_25 )
   END_RUNG
   RUNG wire#w1
      Contact( #In_Functional_Test.Visual_Test_Approved_PLC_Functional_Test_25 )
      Coil( #Out_Functional_Test.Visual_Test_Approved_PLC_Functional_Test_25 )
   END_RUNG
   RUNG wire#w1
      Move(in := #In_Functional_Test.Electrical_Current_Read_PLC_Functional_Test_25, out1 => #Out_Functional_Test.Electrical_Current_Read_PLC_Functional_Test_25)
   END_RUNG
   RUNG wire#w1
      Contact( #In_Functional_Test.Life_Trigger_PLC_Functional_Test_27 )
      Coil( #Out_Functional_Test.Life_Trigger_PLC_Functional_Test_27 )
   END_RUNG
   RUNG wire#w1
      Contact( #In_Functional_Test.Star_Test_PLC_Functional_Test_27 )
      Coil( #Out_Functional_Test.Star_Test_PLC_Functional_Test_27 )
   END_RUNG
   RUNG wire#w1
      Contact( #In_Functional_Test.Button_PLC_Functional_Test_27 )
      Coil( #Out_Functional_Test.Button_PLC_Functional_Test_27 )
   END_RUNG
   RUNG wire#w1
      Contact( #In_Functional_Test.Electrical_Current_Test_Approved_PLC_Functional_Test_27 )
      Coil( #Out_Functional_Test.Electrical_Current_Test_Approved_PLC_Functional_Test_27 )
   END_RUNG
   RUNG wire#w1
      Contact( #In_Functional_Test.Visual_Test_Approved_PLC_Functional_Test_27 )
      Coil( #Out_Functional_Test.Visual_Test_Approved_PLC_Functional_Test_27 )
   END_RUNG
   RUNG wire#w1
      Move(in := #In_Functional_Test.Electrical_Current_Read_PLC_Functional_Test_27, out1 => #Out_Functional_Test.Electrical_Current_Read_PLC_Functional_Test_27)
   END_RUNG
   RUNG wire#w1
      Contact( #In_Functional_Test.Life_Trigger_PLC_Functional_Test_29 )
      Coil( #Out_Functional_Test.Life_Trigger_PLC_Functional_Test_29 )
   END_RUNG
   RUNG wire#w1
      Contact( #In_Functional_Test.Star_Test_PLC_Functional_Test_29 )
      Coil( #Out_Functional_Test.Star_Test_PLC_Functional_Test_29 )
   END_RUNG
   RUNG wire#w1
      Contact( #In_Functional_Test.Button_PLC_Functional_Test_29 )
      Coil( #Out_Functional_Test.Button_PLC_Functional_Test_29 )
   END_RUNG
   RUNG wire#w1
      Contact( #In_Functional_Test.Electrical_Current_Test_Approved_PLC_Functional_Test_29 )
      Coil( #Out_Functional_Test.Electrical_Current_Test_Approved_PLC_Functional_Test_29 )
   END_RUNG
   RUNG wire#w1
      Contact( #In_Functional_Test.Visual_Test_Approved_PLC_Functional_Test_29 )
      Coil( #Out_Functional_Test.Visual_Test_Approved_PLC_Functional_Test_29 )
   END_RUNG
   RUNG wire#w1
      Move(in := #In_Functional_Test.Electrical_Current_Read_PLC_Functional_Test_29, out1 => #Out_Functional_Test.Electrical_Current_Read_PLC_Functional_Test_29)
   END_RUNG
   // the same network as SCL:
   #_w1 := #Test_Station = 13;
   #Out_Functional_Test.Life_Trigger_PLC_Functional_Test_13 := #_w1 AND #Life_Trigger;
   #Out_Functional_Test.Star_Test_PLC_Functional_Test_13 := #_w1 AND #Star_Test;
   #Out_Functional_Test.Button_PLC_Functional_Test_13 := #_w1 AND #Button_Start_Approve;
   #Out_Functional_Test.Electrical_Current_Test_Approved_PLC_Functional_Test_13 := #_w1 AND #Electrical_Current_Test_Approved;
   #Out_Functional_Test.Visual_Test_Approved_PLC_Functional_Test_13 := #_w1 AND #Visual_Test_Approved;
   #Reset_Functional_Test := #_w1 AND #In_Test_Parameters.Reset_PLC_Functional_Test_13;
   IF #_w1 THEN
       #Out_Functional_Test.Electrical_Current_Read_PLC_Functional_Test_13 := #Electrical_Current_Read;
   END_IF;
   #Out_Functional_Test.Life_Trigger_PLC_Functional_Test_15 := #_w1 AND #In_Functional_Test.Life_Trigger_PLC_Functional_Test_15;
   #Out_Functional_Test.Star_Test_PLC_Functional_Test_15 := #_w1 AND #In_Functional_Test.Star_Test_PLC_Functional_Test_15;
   #Out_Functional_Test.Button_PLC_Functional_Test_15 := #_w1 AND #In_Functional_Test.Button_PLC_Functional_Test_15;
   #Out_Functional_Test.Electrical_Current_Test_Approved_PLC_Functional_Test_15 := #_w1 AND #In_Functional_Test.Electrical_Current_Test_Approved_PLC_Functional_Test_15;
   #Out_Functional_Test.Visual_Test_Approved_PLC_Functional_Test_15 := #_w1 AND #In_Functional_Test.Visual_Test_Approved_PLC_Functional_Test_15;
   IF #_w1 THEN
       #Out_Functional_Test.Electrical_Current_Read_PLC_Functional_Test_15 := #In_Functional_Test.Electrical_Current_Read_PLC_Functional_Test_15;
   END_IF;
   #Out_Functional_Test.Life_Trigger_PLC_Functional_Test_17 := #_w1 AND #In_Functional_Test.Life_Trigger_PLC_Functional_Test_17;
   #Out_Functional_Test.Star_Test_PLC_Functional_Test_17 := #_w1 AND #In_Functional_Test.Star_Test_PLC_Functional_Test_17;
   #Out_Functional_Test.Button_PLC_Functional_Test_17 := #_w1 AND #In_Functional_Test.Button_PLC_Functional_Test_17;
   #Out_Functional_Test.Electrical_Current_Test_Approved_PLC_Functional_Test_17 := #_w1 AND #In_Functional_Test.Electrical_Current_Test_Approved_PLC_Functional_Test_17;
   #Out_Functional_Test.Visual_Test_Approved_PLC_Functional_Test_17 := #_w1 AND #In_Functional_Test.Visual_Test_Approved_PLC_Functional_Test_17;
   IF #_w1 THEN
       #Out_Functional_Test.Electrical_Current_Read_PLC_Functional_Test_17 := #In_Functional_Test.Electrical_Current_Read_PLC_Functional_Test_17;
   END_IF;
   #Out_Functional_Test.Life_Trigger_PLC_Functional_Test_19 := #_w1 AND #In_Functional_Test.Life_Trigger_PLC_Functional_Test_19;
   #Out_Functional_Test.Star_Test_PLC_Functional_Test_19 := #_w1 AND #In_Functional_Test.Star_Test_PLC_Functional_Test_19;
   #Out_Functional_Test.Button_PLC_Functional_Test_19 := #_w1 AND #In_Functional_Test.Button_PLC_Functional_Test_19;
   #Out_Functional_Test.Electrical_Current_Test_Approved_PLC_Functional_Test_19 := #_w1 AND #In_Functional_Test.Electrical_Current_Test_Approved_PLC_Functional_Test_19;
   #Out_Functional_Test.Visual_Test_Approved_PLC_Functional_Test_19 := #_w1 AND #In_Functional_Test.Visual_Test_Approved_PLC_Functional_Test_19;
   IF #_w1 THEN
       #Out_Functional_Test.Electrical_Current_Read_PLC_Functional_Test_19 := #In_Functional_Test.Electrical_Current_Read_PLC_Functional_Test_19;
   END_IF;
   #Out_Functional_Test.Life_Trigger_PLC_Functional_Test_21 := #_w1 AND #In_Functional_Test.Life_Trigger_PLC_Functional_Test_21;
   #Out_Functional_Test.Star_Test_PLC_Functional_Test_21 := #_w1 AND #In_Functional_Test.Star_Test_PLC_Functional_Test_21;
   #Out_Functional_Test.Button_PLC_Functional_Test_21 := #_w1 AND #In_Functional_Test.Button_PLC_Functional_Test_21;
   #Out_Functional_Test.Electrical_Current_Test_Approved_PLC_Functional_Test_21 := #_w1 AND #In_Functional_Test.Electrical_Current_Test_Approved_PLC_Functional_Test_21;
   #Out_Functional_Test.Visual_Test_Approved_PLC_Functional_Test_21 := #_w1 AND #In_Functional_Test.Visual_Test_Approved_PLC_Functional_Test_21;
   IF #_w1 THEN
       #Out_Functional_Test.Electrical_Current_Read_PLC_Functional_Test_21 := #In_Functional_Test.Electrical_Current_Read_PLC_Functional_Test_21;
   END_IF;
   #Out_Functional_Test.Life_Trigger_PLC_Functional_Test_23 := #_w1 AND #In_Functional_Test.Life_Trigger_PLC_Functional_Test_23;
   #Out_Functional_Test.Star_Test_PLC_Functional_Test_23 := #_w1 AND #In_Functional_Test.Star_Test_PLC_Functional_Test_23;
   #Out_Functional_Test.Button_PLC_Functional_Test_23 := #_w1 AND #In_Functional_Test.Button_PLC_Functional_Test_23;
   #Out_Functional_Test.Electrical_Current_Test_Approved_PLC_Functional_Test_23 := #_w1 AND #In_Functional_Test.Electrical_Current_Test_Approved_PLC_Functional_Test_23;
   #Out_Functional_Test.Visual_Test_Approved_PLC_Functional_Test_23 := #_w1 AND #In_Functional_Test.Visual_Test_Approved_PLC_Functional_Test_23;
   IF #_w1 THEN
       #Out_Functional_Test.Electrical_Current_Read_PLC_Functional_Test_23 := #In_Functional_Test.Electrical_Current_Read_PLC_Functional_Test_23;
   END_IF;
   #Out_Functional_Test.Life_Trigger_PLC_Functional_Test_25 := #_w1 AND #In_Functional_Test.Life_Trigger_PLC_Functional_Test_25;
   #Out_Functional_Test.Star_Test_PLC_Functional_Test_25 := #_w1 AND #In_Functional_Test.Star_Test_PLC_Functional_Test_25;
   #Out_Functional_Test.Button_PLC_Functional_Test_25 := #_w1 AND #In_Functional_Test.Button_PLC_Functional_Test_25;
   #Out_Functional_Test.Electrical_Current_Test_Approved_PLC_Functional_Test_25 := #_w1 AND #In_Functional_Test.Electrical_Current_Test_Approved_PLC_Functional_Test_25;
   #Out_Functional_Test.Visual_Test_Approved_PLC_Functional_Test_25 := #_w1 AND #In_Functional_Test.Visual_Test_Approved_PLC_Functional_Test_25;
   IF #_w1 THEN
       #Out_Functional_Test.Electrical_Current_Read_PLC_Functional_Test_25 := #In_Functional_Test.Electrical_Current_Read_PLC_Functional_Test_25;
   END_IF;
   #Out_Functional_Test.Life_Trigger_PLC_Functional_Test_27 := #_w1 AND #In_Functional_Test.Life_Trigger_PLC_Functional_Test_27;
   #Out_Functional_Test.Star_Test_PLC_Functional_Test_27 := #_w1 AND #In_Functional_Test.Star_Test_PLC_Functional_Test_27;
   #Out_Functional_Test.Button_PLC_Functional_Test_27 := #_w1 AND #In_Functional_Test.Button_PLC_Functional_Test_27;
   #Out_Functional_Test.Electrical_Current_Test_Approved_PLC_Functional_Test_27 := #_w1 AND #In_Functional_Test.Electrical_Current_Test_Approved_PLC_Functional_Test_27;
   #Out_Functional_Test.Visual_Test_Approved_PLC_Functional_Test_27 := #_w1 AND #In_Functional_Test.Visual_Test_Approved_PLC_Functional_Test_27;
   IF #_w1 THEN
       #Out_Functional_Test.Electrical_Current_Read_PLC_Functional_Test_27 := #In_Functional_Test.Electrical_Current_Read_PLC_Functional_Test_27;
   END_IF;
   #Out_Functional_Test.Life_Trigger_PLC_Functional_Test_29 := #_w1 AND #In_Functional_Test.Life_Trigger_PLC_Functional_Test_29;
   #Out_Functional_Test.Star_Test_PLC_Functional_Test_29 := #_w1 AND #In_Functional_Test.Star_Test_PLC_Functional_Test_29;
   #Out_Functional_Test.Button_PLC_Functional_Test_29 := #_w1 AND #In_Functional_Test.Button_PLC_Functional_Test_29;
   #Out_Functional_Test.Electrical_Current_Test_Approved_PLC_Functional_Test_29 := #_w1 AND #In_Functional_Test.Electrical_Current_Test_Approved_PLC_Functional_Test_29;
   #Out_Functional_Test.Visual_Test_Approved_PLC_Functional_Test_29 := #_w1 AND #In_Functional_Test.Visual_Test_Approved_PLC_Functional_Test_29;
   IF #_w1 THEN
       #Out_Functional_Test.Electrical_Current_Read_PLC_Functional_Test_29 := #In_Functional_Test.Electrical_Current_Read_PLC_Functional_Test_29;
   END_IF;
END_REGION

REGION Network 9: Functional Test Station 15
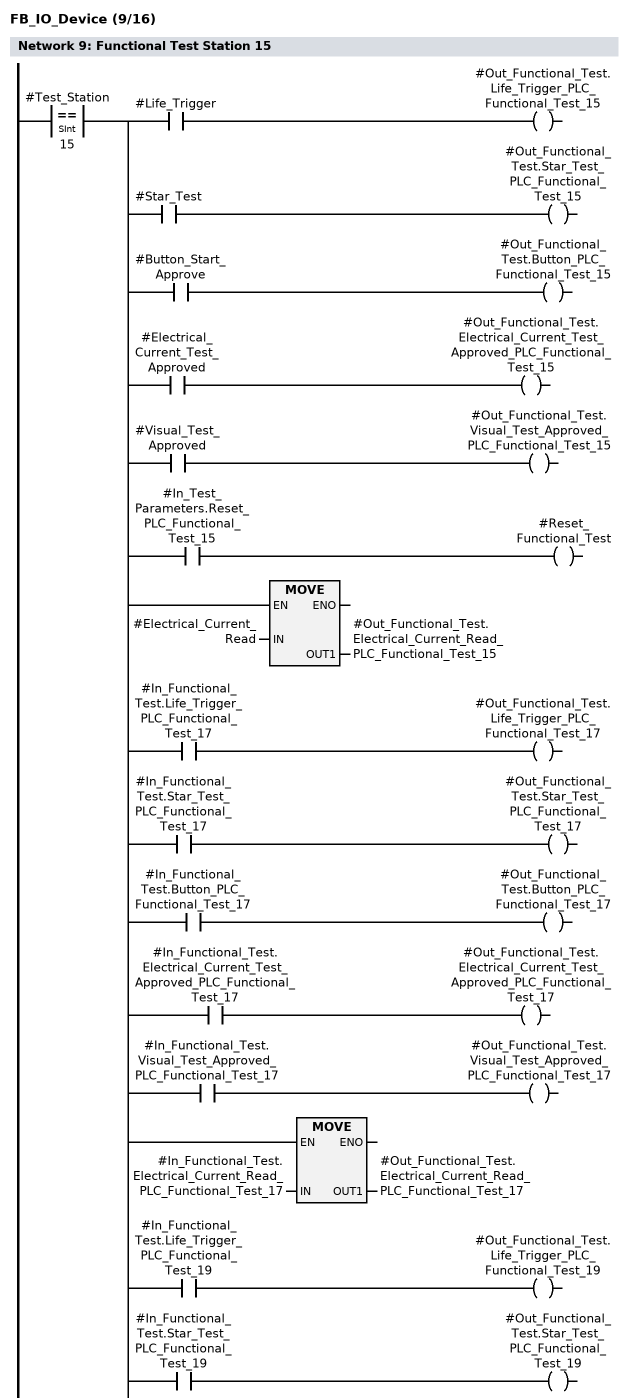
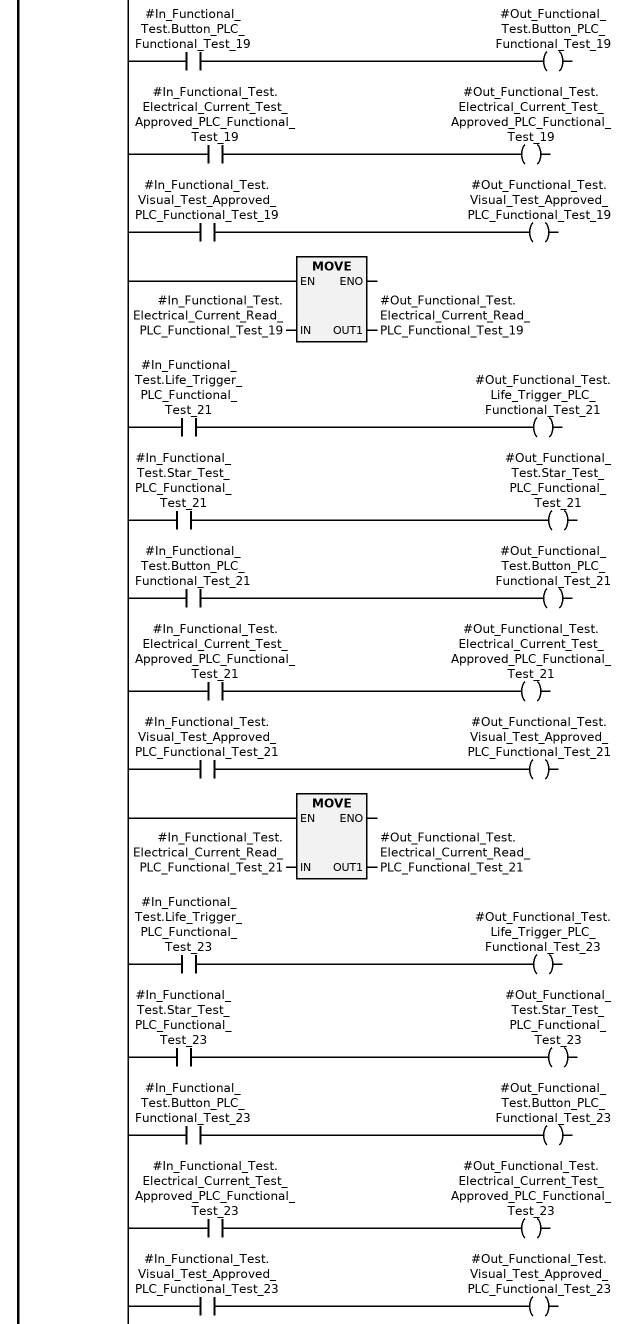
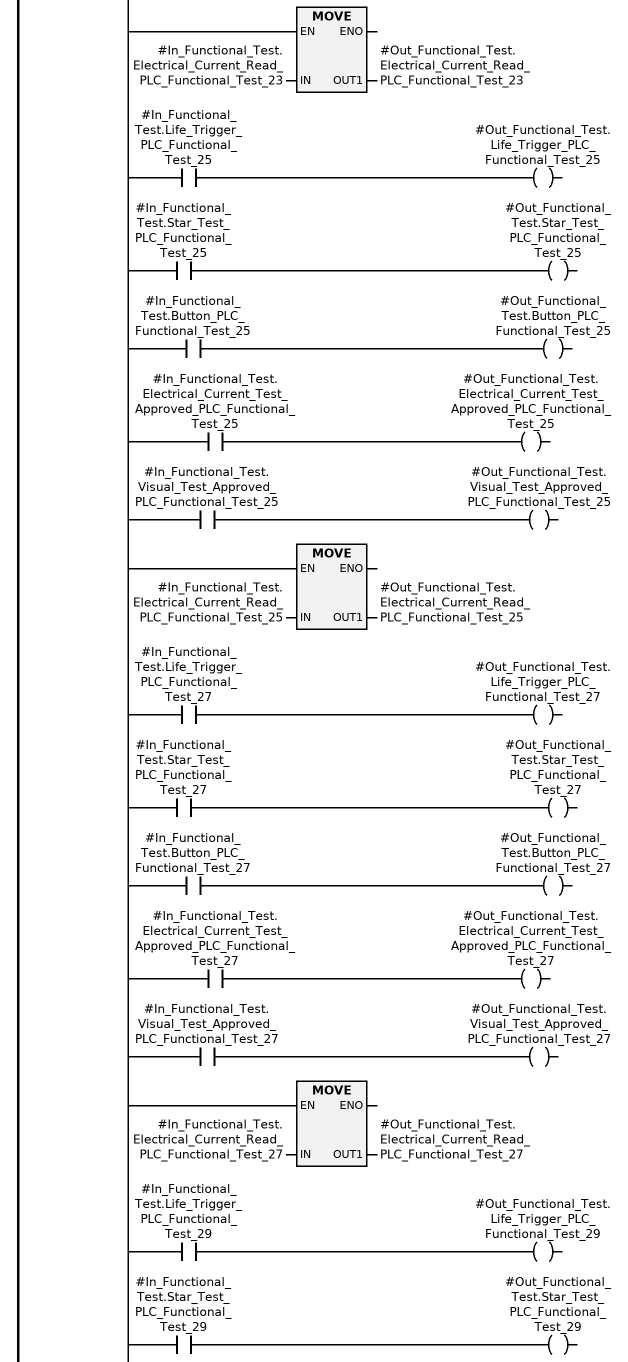
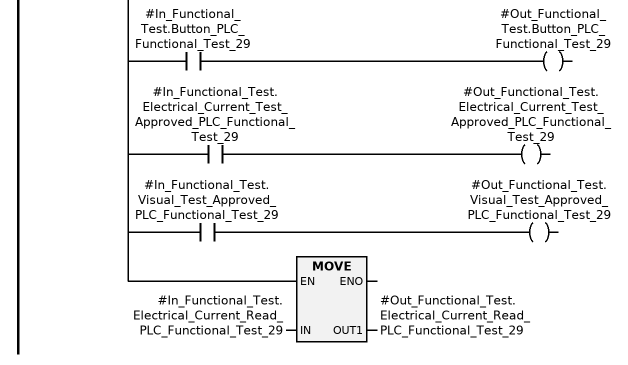
   RUNG wire#powerrail
      { S7_Templates := "SrcType := SInt" } EQ_Contact(in1 := #Test_Station, in2 := 15)
      wire#w1
      Contact( #Life_Trigger )
      Coil( #Out_Functional_Test.Life_Trigger_PLC_Functional_Test_15 )
   END_RUNG
   RUNG wire#w1
      Contact( #Star_Test )
      Coil( #Out_Functional_Test.Star_Test_PLC_Functional_Test_15 )
   END_RUNG
   RUNG wire#w1
      Contact( #Button_Start_Approve )
      Coil( #Out_Functional_Test.Button_PLC_Functional_Test_15 )
   END_RUNG
   RUNG wire#w1
      Contact( #Electrical_Current_Test_Approved )
      Coil( #Out_Functional_Test.Electrical_Current_Test_Approved_PLC_Functional_Test_15 )
   END_RUNG
   RUNG wire#w1
      Contact( #Visual_Test_Approved )
      Coil( #Out_Functional_Test.Visual_Test_Approved_PLC_Functional_Test_15 )
   END_RUNG
   RUNG wire#w1
      Contact( #In_Test_Parameters.Reset_PLC_Functional_Test_15 )
      Coil( #Reset_Functional_Test )
   END_RUNG
   RUNG wire#w1
      Move(in := #Electrical_Current_Read, out1 => #Out_Functional_Test.Electrical_Current_Read_PLC_Functional_Test_15)
   END_RUNG
   RUNG wire#w1
      Contact( #In_Functional_Test.Life_Trigger_PLC_Functional_Test_17 )
      Coil( #Out_Functional_Test.Life_Trigger_PLC_Functional_Test_17 )
   END_RUNG
   RUNG wire#w1
      Contact( #In_Functional_Test.Star_Test_PLC_Functional_Test_17 )
      Coil( #Out_Functional_Test.Star_Test_PLC_Functional_Test_17 )
   END_RUNG
   RUNG wire#w1
      Contact( #In_Functional_Test.Button_PLC_Functional_Test_17 )
      Coil( #Out_Functional_Test.Button_PLC_Functional_Test_17 )
   END_RUNG
   RUNG wire#w1
      Contact( #In_Functional_Test.Electrical_Current_Test_Approved_PLC_Functional_Test_17 )
      Coil( #Out_Functional_Test.Electrical_Current_Test_Approved_PLC_Functional_Test_17 )
   END_RUNG
   RUNG wire#w1
      Contact( #In_Functional_Test.Visual_Test_Approved_PLC_Functional_Test_17 )
      Coil( #Out_Functional_Test.Visual_Test_Approved_PLC_Functional_Test_17 )
   END_RUNG
   RUNG wire#w1
      Move(in := #In_Functional_Test.Electrical_Current_Read_PLC_Functional_Test_17, out1 => #Out_Functional_Test.Electrical_Current_Read_PLC_Functional_Test_17)
   END_RUNG
   RUNG wire#w1
      Contact( #In_Functional_Test.Life_Trigger_PLC_Functional_Test_19 )
      Coil( #Out_Functional_Test.Life_Trigger_PLC_Functional_Test_19 )
   END_RUNG
   RUNG wire#w1
      Contact( #In_Functional_Test.Star_Test_PLC_Functional_Test_19 )
      Coil( #Out_Functional_Test.Star_Test_PLC_Functional_Test_19 )
   END_RUNG
   RUNG wire#w1
      Contact( #In_Functional_Test.Button_PLC_Functional_Test_19 )
      Coil( #Out_Functional_Test.Button_PLC_Functional_Test_19 )
   END_RUNG
   RUNG wire#w1
      Contact( #In_Functional_Test.Electrical_Current_Test_Approved_PLC_Functional_Test_19 )
      Coil( #Out_Functional_Test.Electrical_Current_Test_Approved_PLC_Functional_Test_19 )
   END_RUNG
   RUNG wire#w1
      Contact( #In_Functional_Test.Visual_Test_Approved_PLC_Functional_Test_19 )
      Coil( #Out_Functional_Test.Visual_Test_Approved_PLC_Functional_Test_19 )
   END_RUNG
   RUNG wire#w1
      Move(in := #In_Functional_Test.Electrical_Current_Read_PLC_Functional_Test_19, out1 => #Out_Functional_Test.Electrical_Current_Read_PLC_Functional_Test_19)
   END_RUNG
   RUNG wire#w1
      Contact( #In_Functional_Test.Life_Trigger_PLC_Functional_Test_21 )
      Coil( #Out_Functional_Test.Life_Trigger_PLC_Functional_Test_21 )
   END_RUNG
   RUNG wire#w1
      Contact( #In_Functional_Test.Star_Test_PLC_Functional_Test_21 )
      Coil( #Out_Functional_Test.Star_Test_PLC_Functional_Test_21 )
   END_RUNG
   RUNG wire#w1
      Contact( #In_Functional_Test.Button_PLC_Functional_Test_21 )
      Coil( #Out_Functional_Test.Button_PLC_Functional_Test_21 )
   END_RUNG
   RUNG wire#w1
      Contact( #In_Functional_Test.Electrical_Current_Test_Approved_PLC_Functional_Test_21 )
      Coil( #Out_Functional_Test.Electrical_Current_Test_Approved_PLC_Functional_Test_21 )
   END_RUNG
   RUNG wire#w1
      Contact( #In_Functional_Test.Visual_Test_Approved_PLC_Functional_Test_21 )
      Coil( #Out_Functional_Test.Visual_Test_Approved_PLC_Functional_Test_21 )
   END_RUNG
   RUNG wire#w1
      Move(in := #In_Functional_Test.Electrical_Current_Read_PLC_Functional_Test_21, out1 => #Out_Functional_Test.Electrical_Current_Read_PLC_Functional_Test_21)
   END_RUNG
   RUNG wire#w1
      Contact( #In_Functional_Test.Life_Trigger_PLC_Functional_Test_23 )
      Coil( #Out_Functional_Test.Life_Trigger_PLC_Functional_Test_23 )
   END_RUNG
   RUNG wire#w1
      Contact( #In_Functional_Test.Star_Test_PLC_Functional_Test_23 )
      Coil( #Out_Functional_Test.Star_Test_PLC_Functional_Test_23 )
   END_RUNG
   RUNG wire#w1
      Contact( #In_Functional_Test.Button_PLC_Functional_Test_23 )
      Coil( #Out_Functional_Test.Button_PLC_Functional_Test_23 )
   END_RUNG
   RUNG wire#w1
      Contact( #In_Functional_Test.Electrical_Current_Test_Approved_PLC_Functional_Test_23 )
      Coil( #Out_Functional_Test.Electrical_Current_Test_Approved_PLC_Functional_Test_23 )
   END_RUNG
   RUNG wire#w1
      Contact( #In_Functional_Test.Visual_Test_Approved_PLC_Functional_Test_23 )
      Coil( #Out_Functional_Test.Visual_Test_Approved_PLC_Functional_Test_23 )
   END_RUNG
   RUNG wire#w1
      Move(in := #In_Functional_Test.Electrical_Current_Read_PLC_Functional_Test_23, out1 => #Out_Functional_Test.Electrical_Current_Read_PLC_Functional_Test_23)
   END_RUNG
   RUNG wire#w1
      Contact( #In_Functional_Test.Life_Trigger_PLC_Functional_Test_25 )
      Coil( #Out_Functional_Test.Life_Trigger_PLC_Functional_Test_25 )
   END_RUNG
   RUNG wire#w1
      Contact( #In_Functional_Test.Star_Test_PLC_Functional_Test_25 )
      Coil( #Out_Functional_Test.Star_Test_PLC_Functional_Test_25 )
   END_RUNG
   RUNG wire#w1
      Contact( #In_Functional_Test.Button_PLC_Functional_Test_25 )
      Coil( #Out_Functional_Test.Button_PLC_Functional_Test_25 )
   END_RUNG
   RUNG wire#w1
      Contact( #In_Functional_Test.Electrical_Current_Test_Approved_PLC_Functional_Test_25 )
      Coil( #Out_Functional_Test.Electrical_Current_Test_Approved_PLC_Functional_Test_25 )
   END_RUNG
   RUNG wire#w1
      Contact( #In_Functional_Test.Visual_Test_Approved_PLC_Functional_Test_25 )
      Coil( #Out_Functional_Test.Visual_Test_Approved_PLC_Functional_Test_25 )
   END_RUNG
   RUNG wire#w1
      Move(in := #In_Functional_Test.Electrical_Current_Read_PLC_Functional_Test_25, out1 => #Out_Functional_Test.Electrical_Current_Read_PLC_Functional_Test_25)
   END_RUNG
   RUNG wire#w1
      Contact( #In_Functional_Test.Life_Trigger_PLC_Functional_Test_27 )
      Coil( #Out_Functional_Test.Life_Trigger_PLC_Functional_Test_27 )
   END_RUNG
   RUNG wire#w1
      Contact( #In_Functional_Test.Star_Test_PLC_Functional_Test_27 )
      Coil( #Out_Functional_Test.Star_Test_PLC_Functional_Test_27 )
   END_RUNG
   RUNG wire#w1
      Contact( #In_Functional_Test.Button_PLC_Functional_Test_27 )
      Coil( #Out_Functional_Test.Button_PLC_Functional_Test_27 )
   END_RUNG
   RUNG wire#w1
      Contact( #In_Functional_Test.Electrical_Current_Test_Approved_PLC_Functional_Test_27 )
      Coil( #Out_Functional_Test.Electrical_Current_Test_Approved_PLC_Functional_Test_27 )
   END_RUNG
   RUNG wire#w1
      Contact( #In_Functional_Test.Visual_Test_Approved_PLC_Functional_Test_27 )
      Coil( #Out_Functional_Test.Visual_Test_Approved_PLC_Functional_Test_27 )
   END_RUNG
   RUNG wire#w1
      Move(in := #In_Functional_Test.Electrical_Current_Read_PLC_Functional_Test_27, out1 => #Out_Functional_Test.Electrical_Current_Read_PLC_Functional_Test_27)
   END_RUNG
   RUNG wire#w1
      Contact( #In_Functional_Test.Life_Trigger_PLC_Functional_Test_29 )
      Coil( #Out_Functional_Test.Life_Trigger_PLC_Functional_Test_29 )
   END_RUNG
   RUNG wire#w1
      Contact( #In_Functional_Test.Star_Test_PLC_Functional_Test_29 )
      Coil( #Out_Functional_Test.Star_Test_PLC_Functional_Test_29 )
   END_RUNG
   RUNG wire#w1
      Contact( #In_Functional_Test.Button_PLC_Functional_Test_29 )
      Coil( #Out_Functional_Test.Button_PLC_Functional_Test_29 )
   END_RUNG
   RUNG wire#w1
      Contact( #In_Functional_Test.Electrical_Current_Test_Approved_PLC_Functional_Test_29 )
      Coil( #Out_Functional_Test.Electrical_Current_Test_Approved_PLC_Functional_Test_29 )
   END_RUNG
   RUNG wire#w1
      Contact( #In_Functional_Test.Visual_Test_Approved_PLC_Functional_Test_29 )
      Coil( #Out_Functional_Test.Visual_Test_Approved_PLC_Functional_Test_29 )
   END_RUNG
   RUNG wire#w1
      Move(in := #In_Functional_Test.Electrical_Current_Read_PLC_Functional_Test_29, out1 => #Out_Functional_Test.Electrical_Current_Read_PLC_Functional_Test_29)
   END_RUNG
   // the same network as SCL:
   #_w1 := #Test_Station = 15;
   #Out_Functional_Test.Life_Trigger_PLC_Functional_Test_15 := #_w1 AND #Life_Trigger;
   #Out_Functional_Test.Star_Test_PLC_Functional_Test_15 := #_w1 AND #Star_Test;
   #Out_Functional_Test.Button_PLC_Functional_Test_15 := #_w1 AND #Button_Start_Approve;
   #Out_Functional_Test.Electrical_Current_Test_Approved_PLC_Functional_Test_15 := #_w1 AND #Electrical_Current_Test_Approved;
   #Out_Functional_Test.Visual_Test_Approved_PLC_Functional_Test_15 := #_w1 AND #Visual_Test_Approved;
   #Reset_Functional_Test := #_w1 AND #In_Test_Parameters.Reset_PLC_Functional_Test_15;
   IF #_w1 THEN
       #Out_Functional_Test.Electrical_Current_Read_PLC_Functional_Test_15 := #Electrical_Current_Read;
   END_IF;
   #Out_Functional_Test.Life_Trigger_PLC_Functional_Test_17 := #_w1 AND #In_Functional_Test.Life_Trigger_PLC_Functional_Test_17;
   #Out_Functional_Test.Star_Test_PLC_Functional_Test_17 := #_w1 AND #In_Functional_Test.Star_Test_PLC_Functional_Test_17;
   #Out_Functional_Test.Button_PLC_Functional_Test_17 := #_w1 AND #In_Functional_Test.Button_PLC_Functional_Test_17;
   #Out_Functional_Test.Electrical_Current_Test_Approved_PLC_Functional_Test_17 := #_w1 AND #In_Functional_Test.Electrical_Current_Test_Approved_PLC_Functional_Test_17;
   #Out_Functional_Test.Visual_Test_Approved_PLC_Functional_Test_17 := #_w1 AND #In_Functional_Test.Visual_Test_Approved_PLC_Functional_Test_17;
   IF #_w1 THEN
       #Out_Functional_Test.Electrical_Current_Read_PLC_Functional_Test_17 := #In_Functional_Test.Electrical_Current_Read_PLC_Functional_Test_17;
   END_IF;
   #Out_Functional_Test.Life_Trigger_PLC_Functional_Test_19 := #_w1 AND #In_Functional_Test.Life_Trigger_PLC_Functional_Test_19;
   #Out_Functional_Test.Star_Test_PLC_Functional_Test_19 := #_w1 AND #In_Functional_Test.Star_Test_PLC_Functional_Test_19;
   #Out_Functional_Test.Button_PLC_Functional_Test_19 := #_w1 AND #In_Functional_Test.Button_PLC_Functional_Test_19;
   #Out_Functional_Test.Electrical_Current_Test_Approved_PLC_Functional_Test_19 := #_w1 AND #In_Functional_Test.Electrical_Current_Test_Approved_PLC_Functional_Test_19;
   #Out_Functional_Test.Visual_Test_Approved_PLC_Functional_Test_19 := #_w1 AND #In_Functional_Test.Visual_Test_Approved_PLC_Functional_Test_19;
   IF #_w1 THEN
       #Out_Functional_Test.Electrical_Current_Read_PLC_Functional_Test_19 := #In_Functional_Test.Electrical_Current_Read_PLC_Functional_Test_19;
   END_IF;
   #Out_Functional_Test.Life_Trigger_PLC_Functional_Test_21 := #_w1 AND #In_Functional_Test.Life_Trigger_PLC_Functional_Test_21;
   #Out_Functional_Test.Star_Test_PLC_Functional_Test_21 := #_w1 AND #In_Functional_Test.Star_Test_PLC_Functional_Test_21;
   #Out_Functional_Test.Button_PLC_Functional_Test_21 := #_w1 AND #In_Functional_Test.Button_PLC_Functional_Test_21;
   #Out_Functional_Test.Electrical_Current_Test_Approved_PLC_Functional_Test_21 := #_w1 AND #In_Functional_Test.Electrical_Current_Test_Approved_PLC_Functional_Test_21;
   #Out_Functional_Test.Visual_Test_Approved_PLC_Functional_Test_21 := #_w1 AND #In_Functional_Test.Visual_Test_Approved_PLC_Functional_Test_21;
   IF #_w1 THEN
       #Out_Functional_Test.Electrical_Current_Read_PLC_Functional_Test_21 := #In_Functional_Test.Electrical_Current_Read_PLC_Functional_Test_21;
   END_IF;
   #Out_Functional_Test.Life_Trigger_PLC_Functional_Test_23 := #_w1 AND #In_Functional_Test.Life_Trigger_PLC_Functional_Test_23;
   #Out_Functional_Test.Star_Test_PLC_Functional_Test_23 := #_w1 AND #In_Functional_Test.Star_Test_PLC_Functional_Test_23;
   #Out_Functional_Test.Button_PLC_Functional_Test_23 := #_w1 AND #In_Functional_Test.Button_PLC_Functional_Test_23;
   #Out_Functional_Test.Electrical_Current_Test_Approved_PLC_Functional_Test_23 := #_w1 AND #In_Functional_Test.Electrical_Current_Test_Approved_PLC_Functional_Test_23;
   #Out_Functional_Test.Visual_Test_Approved_PLC_Functional_Test_23 := #_w1 AND #In_Functional_Test.Visual_Test_Approved_PLC_Functional_Test_23;
   IF #_w1 THEN
       #Out_Functional_Test.Electrical_Current_Read_PLC_Functional_Test_23 := #In_Functional_Test.Electrical_Current_Read_PLC_Functional_Test_23;
   END_IF;
   #Out_Functional_Test.Life_Trigger_PLC_Functional_Test_25 := #_w1 AND #In_Functional_Test.Life_Trigger_PLC_Functional_Test_25;
   #Out_Functional_Test.Star_Test_PLC_Functional_Test_25 := #_w1 AND #In_Functional_Test.Star_Test_PLC_Functional_Test_25;
   #Out_Functional_Test.Button_PLC_Functional_Test_25 := #_w1 AND #In_Functional_Test.Button_PLC_Functional_Test_25;
   #Out_Functional_Test.Electrical_Current_Test_Approved_PLC_Functional_Test_25 := #_w1 AND #In_Functional_Test.Electrical_Current_Test_Approved_PLC_Functional_Test_25;
   #Out_Functional_Test.Visual_Test_Approved_PLC_Functional_Test_25 := #_w1 AND #In_Functional_Test.Visual_Test_Approved_PLC_Functional_Test_25;
   IF #_w1 THEN
       #Out_Functional_Test.Electrical_Current_Read_PLC_Functional_Test_25 := #In_Functional_Test.Electrical_Current_Read_PLC_Functional_Test_25;
   END_IF;
   #Out_Functional_Test.Life_Trigger_PLC_Functional_Test_27 := #_w1 AND #In_Functional_Test.Life_Trigger_PLC_Functional_Test_27;
   #Out_Functional_Test.Star_Test_PLC_Functional_Test_27 := #_w1 AND #In_Functional_Test.Star_Test_PLC_Functional_Test_27;
   #Out_Functional_Test.Button_PLC_Functional_Test_27 := #_w1 AND #In_Functional_Test.Button_PLC_Functional_Test_27;
   #Out_Functional_Test.Electrical_Current_Test_Approved_PLC_Functional_Test_27 := #_w1 AND #In_Functional_Test.Electrical_Current_Test_Approved_PLC_Functional_Test_27;
   #Out_Functional_Test.Visual_Test_Approved_PLC_Functional_Test_27 := #_w1 AND #In_Functional_Test.Visual_Test_Approved_PLC_Functional_Test_27;
   IF #_w1 THEN
       #Out_Functional_Test.Electrical_Current_Read_PLC_Functional_Test_27 := #In_Functional_Test.Electrical_Current_Read_PLC_Functional_Test_27;
   END_IF;
   #Out_Functional_Test.Life_Trigger_PLC_Functional_Test_29 := #_w1 AND #In_Functional_Test.Life_Trigger_PLC_Functional_Test_29;
   #Out_Functional_Test.Star_Test_PLC_Functional_Test_29 := #_w1 AND #In_Functional_Test.Star_Test_PLC_Functional_Test_29;
   #Out_Functional_Test.Button_PLC_Functional_Test_29 := #_w1 AND #In_Functional_Test.Button_PLC_Functional_Test_29;
   #Out_Functional_Test.Electrical_Current_Test_Approved_PLC_Functional_Test_29 := #_w1 AND #In_Functional_Test.Electrical_Current_Test_Approved_PLC_Functional_Test_29;
   #Out_Functional_Test.Visual_Test_Approved_PLC_Functional_Test_29 := #_w1 AND #In_Functional_Test.Visual_Test_Approved_PLC_Functional_Test_29;
   IF #_w1 THEN
       #Out_Functional_Test.Electrical_Current_Read_PLC_Functional_Test_29 := #In_Functional_Test.Electrical_Current_Read_PLC_Functional_Test_29;
   END_IF;
END_REGION

